LIN {X 0,Y 523.905,Z 250.039,A -85,B 0,C 180,E1 -4666.027,E2 -4666.027} C_VEL
LIN {X 0,Y 523.954,Z 250.034,A -85,B 0,C 180,E1 -4668.393,E2 -4668.393} C_VEL
LIN {X 0,Y 523.94,Z 250.032,A -85,B 0,C 180,E1 -4671.515,E2 -4671.515} C_VEL
LIN {X 0,Y 524.027,Z 250.021,A -85,B 0,C 180,E1 -4674.613,E2 -4674.613} C_VEL
LIN {X 0,Y 524.098,Z 250.015,A -85,B 0,C 180,E1 -4677.694,E2 -4677.694} C_VEL
LIN {X 0,Y 524.09,Z 250.017,A -85,B 0,C 180,E1 -4680,E2 -4680} C_VEL
LIN {X 0,Y 524.098,Z 250.013,A -85,B 0,C 180,E1 -4682.305,E2 -4682.305} C_VEL
LIN {X 0,Y 523.995,Z 250.027,A -85,B 0,C 180,E1 -4686.16,E2 -4686.16} C_VEL
LIN {X 0,Y 523.937,Z 250.033,A -85,B 0,C 180,E1 -4689.263,E2 -4689.263} C_VEL
LIN {X 0,Y 523.937,Z 250.031,A -85,B 0,C 180,E1 -4692.393,E2 -4692.393} C_VEL
LIN {X 0,Y 523.905,Z 250.04,A -85,B 0,C 180,E1 -4695.563,E2 -4695.563} C_VEL
LIN {X 0,Y 523.903,Z 250.037,A -85,B 0,C 180,E1 -4697.971,E2 -4697.971} C_VEL
LIN {X 0,Y 523.909,Z 250.033,A -85,B 0,C 180,E1 -4700.412,E2 -4700.412} C_VEL
LIN {X 0,Y 523.878,Z 250.039,A -85,B 0,C 180,E1 -4702.895,E2 -4702.895} C_VEL
LIN {X 0,Y 523.889,Z 250.043,A -85,B 0,C 180,E1 -4705.422,E2 -4705.422} C_VEL
LIN {X 0,Y 523.889,Z 250.037,A -85,B 0,C 180,E1 -4708.003,E2 -4708.003} C_VEL
LIN {X 0,Y 523.891,Z 250.039,A -85,B 0,C 180,E1 -4710.846,E2 -4710.846} C_VEL
LIN {X 0,Y 523.92,Z 250.034,A -85,B 0,C 180,E1 -4713.729,E2 -4713.729} C_VEL
LIN {X 0,Y 523.861,Z 250.04,A -85,B 0,C 180,E1 -4716.396,E2 -4716.396} C_VEL
LIN {X 0,Y 523.897,Z 250.042,A -85,B 0,C 180,E1 -4719.087,E2 -4719.087} C_VEL
LIN {X 0,Y 523.887,Z 250.036,A -85,B 0,C 180,E1 -4722.125,E2 -4722.125} C_VEL
LIN {X 0,Y 523.928,Z 250.035,A -85,B 0,C 180,E1 -4725.312,E2 -4725.312} C_VEL
LIN {X 0,Y 523.906,Z 250.038,A -85,B 0,C 180,E1 -4728.696,E2 -4728.696} C_VEL
LIN {X 0,Y 523.894,Z 250.035,A -85,B 0,C 180,E1 -4731.897,E2 -4731.897} C_VEL
LIN {X 0,Y 523.906,Z 250.04,A -85,B 0,C 180,E1 -4734.914,E2 -4734.914} C_VEL
LIN {X 0,Y 523.894,Z 250.034,A -85,B 0,C 180,E1 -4737.687,E2 -4737.687} C_VEL
LIN {X 0,Y 523.861,Z 250.041,A -85,B 0,C 180,E1 -4740.24,E2 -4740.24} C_VEL
LIN {X 0,Y 523.887,Z 250.042,A -85,B 0,C 180,E1 -4742.864,E2 -4742.864} C_VEL
LIN {X 0,Y 523.92,Z 250.04,A -85,B 0,C 180,E1 -4746.271,E2 -4746.271} C_VEL
LIN {X 0,Y 524.919,Z 256.867,A -85,B 0,C 180,E1 -4747.491,E2 -4747.491} C_VEL
LIN {X 0,Y 524.608,Z 272.008,A -85,B 0,C 180,E1 -4750.04,E2 -4750.04} C_VEL
LIN {X 0,Y 524.347,Z 287.74,A -85,B 0,C 180,E1 -4752.658,E2 -4752.658} C_VEL
LIN {X 0,Y 524.067,Z 307.036,A -85,B 0,C 180,E1 -4755.834,E2 -4755.834} C_VEL
LIN {X 0,Y 523.837,Z 320.787,A -85,B 0,C 180,E1 -4758.077,E2 -4758.077} C_VEL
LIN {X 0,Y 524.912,Z 332.835,A -85,B 0,C 180,E1 -4758.269,E2 -4758.269} C_VEL
LIN {X 0,Y 524.717,Z 397.742,A -85,B 0,C 180,E1 -4759.168,E2 -4759.168} C_VEL
LIN {X 0,Y 524.544,Z 407.017,A -85,B 0,C 180,E1 -4759.384,E2 -4759.384} C_VEL
LIN {X 0,Y 524.443,Z 415.51,A -85,B 0,C 180,E1 -4759.675,E2 -4759.675} C_VEL
LIN {X 0,Y 524.283,Z 424.041,A -85,B 0,C 180,E1 -4760.062,E2 -4760.062} C_VEL
LIN {X 0,Y 524.146,Z 432.41,A -85,B 0,C 180,E1 -4760.547,E2 -4760.547} C_VEL
LIN {X 0,Y 524.027,Z 440.49,A -85,B 0,C 180,E1 -4761.128,E2 -4761.128} C_VEL
LIN {X 0,Y 523.808,Z 449.21,A -85,B 0,C 180,E1 -4761.902,E2 -4761.902} C_VEL
LIN {X 0,Y 523.696,Z 457.778,A -85,B 0,C 180,E1 -4762.87,E2 -4762.87} C_VEL
LIN {X 0,Y 523.586,Z 464.502,A -85,B 0,C 180,E1 -4763.836,E2 -4763.836} C_VEL
LIN {X 0,Y 523.483,Z 468.916,A -85,B 0,C 180,E1 -4764.608,E2 -4764.608} C_VEL
LIN {X 0,Y 523.45,Z 474.125,A -85,B 0,C 180,E1 -4765.766,E2 -4765.766} C_VEL
LIN {X 0,Y 523.406,Z 476.787,A -85,B 0,C 180,E1 -4766.536,E2 -4766.536} C_VEL
LIN {X 0,Y 523.336,Z 479.706,A -85,B 0,C 180,E1 -4767.691,E2 -4767.691} C_VEL
LIN {X 0,Y 523.273,Z 480.964,A -85,B 0,C 180,E1 -4768.461,E2 -4768.461} C_VEL
LIN {X 0,Y 523.26,Z 481.749,A -85,B 0,C 180,E1 -4769.231,E2 -4769.231} C_VEL
LIN {X 0,Y 523.264,Z 482.046,A -85,B 0,C 180,E1 -4770,E2 -4770} C_VEL
LIN {X 0,Y 523.26,Z 481.748,A -85,B 0,C 180,E1 -4770.77,E2 -4770.77} C_VEL
LIN {X 0,Y 523.273,Z 480.963,A -85,B 0,C 180,E1 -4771.54,E2 -4771.54} C_VEL
LIN {X 0,Y 523.336,Z 479.704,A -85,B 0,C 180,E1 -4772.309,E2 -4772.309} C_VEL
LIN {X 0,Y 523.407,Z 476.784,A -85,B 0,C 180,E1 -4773.464,E2 -4773.464} C_VEL
LIN {X 0,Y 523.451,Z 474.122,A -85,B 0,C 180,E1 -4774.235,E2 -4774.235} C_VEL
LIN {X 0,Y 523.483,Z 468.909,A -85,B 0,C 180,E1 -4775.393,E2 -4775.393} C_VEL
LIN {X 0,Y 523.573,Z 462.995,A -85,B 0,C 180,E1 -4776.409,E2 -4776.409} C_VEL
LIN {X 0,Y 523.699,Z 456.256,A -85,B 0,C 180,E1 -4777.325,E2 -4777.325} C_VEL
LIN {X 0,Y 523.833,Z 448.182,A -85,B 0,C 180,E1 -4778.196,E2 -4778.196} C_VEL
LIN {X 0,Y 524.028,Z 440.484,A -85,B 0,C 180,E1 -4778.873,E2 -4778.873} C_VEL
LIN {X 0,Y 524.147,Z 432.399,A -85,B 0,C 180,E1 -4779.454,E2 -4779.454} C_VEL
LIN {X 0,Y 524.283,Z 424.028,A -85,B 0,C 180,E1 -4779.939,E2 -4779.939} C_VEL
LIN {X 0,Y 524.443,Z 415.494,A -85,B 0,C 180,E1 -4780.326,E2 -4780.326} C_VEL
LIN {X 0,Y 524.588,Z 405.328,A -85,B 0,C 180,E1 -4780.664,E2 -4780.664} C_VEL
LIN {X 0,Y 524.728,Z 393.603,A -85,B 0,C 180,E1 -4780.906,E2 -4780.906} C_VEL
LIN {X 0,Y 524.84,Z 329.868,A -85,B 0,C 180,E1 -4781.773,E2 -4781.773} C_VEL
LIN {X 0,Y 523.822,Z 320.739,A -85,B 0,C 180,E1 -4781.931,E2 -4781.931} C_VEL
LIN {X 0,Y 524.065,Z 303.407,A -85,B 0,C 180,E1 -4784.762,E2 -4784.762} C_VEL
LIN {X 0,Y 524.416,Z 284.047,A -85,B 0,C 180,E1 -4787.953,E2 -4787.953} C_VEL
LIN {X 0,Y 524.723,Z 265.839,A -85,B 0,C 180,E1 -4790.995,E2 -4790.995} C_VEL
LIN {X 0,Y 524.885,Z 256.204,A -85,B 0,C 180,E1 -4792.623,E2 -4792.623} C_VEL
LIN {X 0,Y 523.923,Z 250.038,A -85,B 0,C 180,E1 -4793.73,E2 -4793.73} C_VEL
LIN {X 0,Y 523.89,Z 250.042,A -85,B 0,C 180,E1 -4797.137,E2 -4797.137} C_VEL
LIN {X 0,Y 523.865,Z 250.041,A -85,B 0,C 180,E1 -4799.761,E2 -4799.761} C_VEL
LIN {X 0,Y 523.895,Z 250.034,A -85,B 0,C 180,E1 -4802.453,E2 -4802.453} C_VEL
LIN {X 0,Y 523.88,Z 250.045,A -85,B 0,C 180,E1 -4805.23,E2 -4805.23} C_VEL
LIN {X 0,Y 523.877,Z 250.037,A -85,B 0,C 180,E1 -4808.105,E2 -4808.105} C_VEL
LIN {X 0,Y 523.88,Z 250.042,A -85,B 0,C 180,E1 -4811.301,E2 -4811.301} C_VEL
LIN {X 0,Y 523.932,Z 250.034,A -85,B 0,C 180,E1 -4814.689,E2 -4814.689} C_VEL
LIN {X 0,Y 523.889,Z 250.035,A -85,B 0,C 180,E1 -4817.875,E2 -4817.875} C_VEL
LIN {X 0,Y 523.894,Z 250.042,A -85,B 0,C 180,E1 -4820.913,E2 -4820.913} C_VEL
LIN {X 0,Y 523.853,Z 250.04,A -85,B 0,C 180,E1 -4823.822,E2 -4823.822} C_VEL
LIN {X 0,Y 523.895,Z 250.041,A -85,B 0,C 180,E1 -4826.632,E2 -4826.632} C_VEL
LIN {X 0,Y 523.906,Z 250.035,A -85,B 0,C 180,E1 -4829.353,E2 -4829.353} C_VEL
LIN {X 0,Y 523.911,Z 250.037,A -85,B 0,C 180,E1 -4832.296,E2 -4832.296} C_VEL
LIN {X 0,Y 523.89,Z 250.036,A -85,B 0,C 180,E1 -4835.426,E2 -4835.426} C_VEL
LIN {X 0,Y 523.92,Z 250.033,A -85,B 0,C 180,E1 -4837.939,E2 -4837.939} C_VEL
LIN {X 0,Y 523.9,Z 250.042,A -85,B 0,C 180,E1 -4840.405,E2 -4840.405} C_VEL
LIN {X 0,Y 523.9,Z 250.038,A -85,B 0,C 180,E1 -4842.835,E2 -4842.835} C_VEL
LIN {X 0,Y 523.92,Z 250.032,A -85,B 0,C 180,E1 -4845.234,E2 -4845.234} C_VEL
LIN {X 0,Y 523.96,Z 250.033,A -85,B 0,C 180,E1 -4848.393,E2 -4848.393} C_VEL
LIN {X 0,Y 523.945,Z 250.03,A -85,B 0,C 180,E1 -4851.515,E2 -4851.515} C_VEL
LIN {X 0,Y 524.028,Z 250.023,A -85,B 0,C 180,E1 -4854.613,E2 -4854.613} C_VEL
LIN {X 0,Y 524.103,Z 250.012,A -85,B 0,C 180,E1 -4857.695,E2 -4857.695} C_VEL
LIN {X 0,Y 524.096,Z 250.017,A -85,B 0,C 180,E1 -4860,E2 -4860} C_VEL
LIN {X 0,Y 524.103,Z 250.014,A -85,B 0,C 180,E1 -4862.306,E2 -4862.306} C_VEL
LIN {X 0,Y 524.001,Z 250.027,A -85,B 0,C 180,E1 -4866.16,E2 -4866.16} C_VEL
LIN {X 0,Y 523.944,Z 250.031,A -85,B 0,C 180,E1 -4869.263,E2 -4869.263} C_VEL
LIN {X 0,Y 523.945,Z 250.032,A -85,B 0,C 180,E1 -4872.393,E2 -4872.393} C_VEL
LIN {X 0,Y 523.913,Z 250.039,A -85,B 0,C 180,E1 -4875.563,E2 -4875.563} C_VEL
LIN {X 0,Y 523.911,Z 250.039,A -85,B 0,C 180,E1 -4877.971,E2 -4877.971} C_VEL
LIN {X 0,Y 523.917,Z 250.034,A -85,B 0,C 180,E1 -4880.412,E2 -4880.412} C_VEL
LIN {X 0,Y 523.885,Z 250.038,A -85,B 0,C 180,E1 -4882.895,E2 -4882.895} C_VEL
LIN {X 0,Y 523.899,Z 250.041,A -85,B 0,C 180,E1 -4885.422,E2 -4885.422} C_VEL
LIN {X 0,Y 523.897,Z 250.038,A -85,B 0,C 180,E1 -4888.003,E2 -4888.003} C_VEL
LIN {X 0,Y 523.902,Z 250.036,A -85,B 0,C 180,E1 -4890.846,E2 -4890.846} C_VEL
LIN {X 0,Y 523.927,Z 250.036,A -85,B 0,C 180,E1 -4893.729,E2 -4893.729} C_VEL
LIN {X 0,Y 523.888,Z 250.037,A -85,B 0,C 180,E1 -4896.399,E2 -4896.399} C_VEL
LIN {X 0,Y 523.91,Z 250.039,A -85,B 0,C 180,E1 -4899.086,E2 -4899.086} C_VEL
LIN {X 0,Y 523.893,Z 250.036,A -85,B 0,C 180,E1 -4902.125,E2 -4902.125} C_VEL
LIN {X 0,Y 523.935,Z 250.036,A -85,B 0,C 180,E1 -4905.311,E2 -4905.311} C_VEL
LIN {X 0,Y 523.879,Z 250.042,A -85,B 0,C 180,E1 -4906.868,E2 -4906.868} C_VEL
LIN {X 0,Y 523.192,Z 250.127,A -85,B 0,C 180,E1 -4907.51,E2 -4907.51} C_VEL
LIN {X 0,Y 520.329,Z 250.482,A -85,B 0,C 180,E1 -4908.551,E2 -4908.551} C_VEL
LIN {X 0,Y 517.935,Z 250.783,A -85,B 0,C 180,E1 -4909.39,E2 -4909.39} C_VEL
LIN {X 0,Y 516.929,Z 250.904,A -85,B 0,C 180,E1 -4910.038,E2 -4910.038} C_VEL
LIN {X 0,Y 516.858,Z 250.913,A -85,B 0,C 180,E1 -4910.257,E2 -4910.257} C_VEL
LIN {X 0,Y 516.854,Z 250.919,A -85,B 0,C 180,E1 -4913.252,E2 -4913.252} C_VEL
LIN {X 0,Y 516.881,Z 250.91,A -85,B 0,C 180,E1 -4916.118,E2 -4916.118} C_VEL
LIN {X 0,Y 516.85,Z 250.919,A -85,B 0,C 180,E1 -4918.944,E2 -4918.944} C_VEL
LIN {X 0,Y 516.846,Z 250.915,A -85,B 0,C 180,E1 -4921.58,E2 -4921.58} C_VEL
LIN {X 0,Y 516.871,Z 250.912,A -85,B 0,C 180,E1 -4924.207,E2 -4924.207} C_VEL
LIN {X 0,Y 516.853,Z 250.918,A -85,B 0,C 180,E1 -4926.775,E2 -4926.775} C_VEL
LIN {X 0,Y 516.929,Z 250.903,A -85,B 0,C 180,E1 -4929.735,E2 -4929.735} C_VEL
LIN {X 0,Y 516.879,Z 250.917,A -85,B 0,C 180,E1 -4932.594,E2 -4932.594} C_VEL
LIN {X 0,Y 516.693,Z 250.994,A -85,B 0,C 180,E1 -4934.548,E2 -4934.548} C_VEL
LIN {X 0,Y 516.644,Z 265.328,A -85,B 0,C 180,E1 -4937.788,E2 -4937.788} C_VEL
LIN {X 0,Y 516.655,Z 266.191,A -85,B 0,C 180,E1 -4937.977,E2 -4937.977} C_VEL
LIN {X 0,Y 518.082,Z 276.255,A -85,B 0,C 180,E1 -4938.154,E2 -4938.154} C_VEL
LIN {X 0,Y 517.773,Z 341.417,A -85,B 0,C 180,E1 -4939.07,E2 -4939.07} C_VEL
LIN {X 0,Y 517.698,Z 349.767,A -85,B 0,C 180,E1 -4939.266,E2 -4939.266} C_VEL
LIN {X 0,Y 517.58,Z 359.014,A -85,B 0,C 180,E1 -4939.585,E2 -4939.585} C_VEL
LIN {X 0,Y 517.478,Z 366.536,A -85,B 0,C 180,E1 -4939.929,E2 -4939.929} C_VEL
LIN {X 0,Y 517.334,Z 375.007,A -85,B 0,C 180,E1 -4940.42,E2 -4940.42} C_VEL
LIN {X 0,Y 517.215,Z 383.133,A -85,B 0,C 180,E1 -4941.01,E2 -4941.01} C_VEL
LIN {X 0,Y 517.03,Z 390.845,A -85,B 0,C 180,E1 -4941.696,E2 -4941.696} C_VEL
LIN {X 0,Y 516.857,Z 397.209,A -85,B 0,C 180,E1 -4942.381,E2 -4942.381} C_VEL
LIN {X 0,Y 516.724,Z 404.187,A -85,B 0,C 180,E1 -4943.293,E2 -4943.293} C_VEL
LIN {X 0,Y 516.5,Z 410.57,A -85,B 0,C 180,E1 -4944.338,E2 -4944.338} C_VEL
LIN {X 0,Y 516.512,Z 415.188,A -85,B 0,C 180,E1 -4945.317,E2 -4945.317} C_VEL
LIN {X 0,Y 516.391,Z 418.177,A -85,B 0,C 180,E1 -4946.098,E2 -4946.098} C_VEL
LIN {X 0,Y 516.403,Z 420.488,A -85,B 0,C 180,E1 -4946.879,E2 -4946.879} C_VEL
LIN {X 0,Y 516.269,Z 422.26,A -85,B 0,C 180,E1 -4947.659,E2 -4947.659} C_VEL
LIN {X 0,Y 516.2,Z 423.537,A -85,B 0,C 180,E1 -4948.439,E2 -4948.439} C_VEL
LIN {X 0,Y 516.186,Z 424.345,A -85,B 0,C 180,E1 -4949.219,E2 -4949.219} C_VEL
LIN {X 0,Y 516.186,Z 424.653,A -85,B 0,C 180,E1 -4950,E2 -4950} C_VEL
LIN {X 0,Y 516.186,Z 424.383,A -85,B 0,C 180,E1 -4950.78,E2 -4950.78} C_VEL
LIN {X 0,Y 516.201,Z 423.649,A -85,B 0,C 180,E1 -4951.56,E2 -4951.56} C_VEL
LIN {X 0,Y 516.269,Z 422.447,A -85,B 0,C 180,E1 -4952.34,E2 -4952.34} C_VEL
LIN {X 0,Y 516.418,Z 419.614,A -85,B 0,C 180,E1 -4953.511,E2 -4953.511} C_VEL
LIN {X 0,Y 516.433,Z 417.043,A -85,B 0,C 180,E1 -4954.292,E2 -4954.292} C_VEL
LIN {X 0,Y 516.433,Z 411.976,A -85,B 0,C 180,E1 -4955.466,E2 -4955.466} C_VEL
LIN {X 0,Y 516.703,Z 405.867,A -85,B 0,C 180,E1 -4956.55,E2 -4956.55} C_VEL
LIN {X 0,Y 516.854,Z 397.988,A -85,B 0,C 180,E1 -4957.618,E2 -4957.618} C_VEL
LIN {X 0,Y 516.995,Z 390.762,A -85,B 0,C 180,E1 -4958.403,E2 -4958.403} C_VEL
LIN {X 0,Y 517.203,Z 384.256,A -85,B 0,C 180,E1 -4958.99,E2 -4958.99} C_VEL
LIN {X 0,Y 517.3,Z 376.382,A -85,B 0,C 180,E1 -4959.58,E2 -4959.58} C_VEL
LIN {X 0,Y 517.484,Z 368.247,A -85,B 0,C 180,E1 -4960.07,E2 -4960.07} C_VEL
LIN {X 0,Y 517.611,Z 360.017,A -85,B 0,C 180,E1 -4960.463,E2 -4960.463} C_VEL
LIN {X 0,Y 517.677,Z 351.151,A -85,B 0,C 180,E1 -4960.783,E2 -4960.783} C_VEL
LIN {X 0,Y 517.866,Z 342.414,A -85,B 0,C 180,E1 -4960.999,E2 -4960.999} C_VEL
LIN {X 0,Y 518.009,Z 295.646,A -85,B 0,C 180,E1 -4961.669,E2 -4961.669} C_VEL
LIN {X 0,Y 518.006,Z 274.632,A -85,B 0,C 180,E1 -4961.961,E2 -4961.961} C_VEL
LIN {X 0,Y 516.658,Z 266.136,A -85,B 0,C 180,E1 -4962.127,E2 -4962.127} C_VEL
LIN {X 0,Y 516.663,Z 251.854,A -85,B 0,C 180,E1 -4965.341,E2 -4965.341} C_VEL
LIN {X 0,Y 516.672,Z 250.945,A -85,B 0,C 180,E1 -4965.563,E2 -4965.563} C_VEL
LIN {X 0,Y 516.873,Z 250.914,A -85,B 0,C 180,E1 -4967.861,E2 -4967.861} C_VEL
LIN {X 0,Y 516.889,Z 250.909,A -85,B 0,C 180,E1 -4970.702,E2 -4970.702} C_VEL
LIN {X 0,Y 516.838,Z 250.921,A -85,B 0,C 180,E1 -4973.224,E2 -4973.224} C_VEL
LIN {X 0,Y 516.879,Z 250.91,A -85,B 0,C 180,E1 -4976.181,E2 -4976.181} C_VEL
LIN {X 0,Y 516.895,Z 250.913,A -85,B 0,C 180,E1 -4979.306,E2 -4979.306} C_VEL
LIN {X 0,Y 516.889,Z 250.91,A -85,B 0,C 180,E1 -4982.542,E2 -4982.542} C_VEL
LIN {X 0,Y 516.851,Z 250.918,A -85,B 0,C 180,E1 -4985.327,E2 -4985.327} C_VEL
LIN {X 0,Y 516.874,Z 250.911,A -85,B 0,C 180,E1 -4987.942,E2 -4987.942} C_VEL
LIN {X 0,Y 516.846,Z 250.92,A -85,B 0,C 180,E1 -4990.744,E2 -4990.744} C_VEL
LIN {X 0,Y 516.876,Z 250.91,A -85,B 0,C 180,E1 -4993.903,E2 -4993.903} C_VEL
LIN {X 0,Y 516.876,Z 250.911,A -85,B 0,C 180,E1 -4996.107,E2 -4996.107} C_VEL
LIN {X 0,Y 516.843,Z 250.917,A -85,B 0,C 180,E1 -4999.254,E2 -4999.254} C_VEL
LIN {X 0,Y 516.871,Z 250.912,A -85,B 0,C 180,E1 -5002.057,E2 -5002.057} C_VEL
LIN {X 0,Y 516.866,Z 250.914,A -85,B 0,C 180,E1 -5005.174,E2 -5005.174} C_VEL
LIN {X 0,Y 516.861,Z 250.913,A -85,B 0,C 180,E1 -5007.974,E2 -5007.974} C_VEL
LIN {X 0,Y 516.892,Z 250.913,A -85,B 0,C 180,E1 -5010.694,E2 -5010.694} C_VEL
LIN {X 0,Y 516.874,Z 250.912,A -85,B 0,C 180,E1 -5013.818,E2 -5013.818} C_VEL
LIN {X 0,Y 516.836,Z 250.919,A -85,B 0,C 180,E1 -5016.775,E2 -5016.775} C_VEL
LIN {X 0,Y 516.901,Z 250.909,A -85,B 0,C 180,E1 -5019.742,E2 -5019.742} C_VEL
LIN {X 0,Y 516.873,Z 250.915,A -85,B 0,C 180,E1 -5022.594,E2 -5022.594} C_VEL
LIN {X 0,Y 516.925,Z 250.905,A -85,B 0,C 180,E1 -5025.03,E2 -5025.03} C_VEL
LIN {X 0,Y 516.92,Z 250.91,A -85,B 0,C 180,E1 -5028.233,E2 -5028.233} C_VEL
LIN {X 0,Y 516.914,Z 250.906,A -85,B 0,C 180,E1 -5031.399,E2 -5031.399} C_VEL
LIN {X 0,Y 516.978,Z 250.9,A -85,B 0,C 180,E1 -5034.539,E2 -5034.539} C_VEL
LIN {X 0,Y 517.067,Z 250.891,A -85,B 0,C 180,E1 -5037.663,E2 -5037.663} C_VEL
LIN {X 0,Y 517.059,Z 250.893,A -85,B 0,C 180,E1 -5040,E2 -5040} C_VEL
LIN {X 0,Y 517.067,Z 250.889,A -85,B 0,C 180,E1 -5042.337,E2 -5042.337} C_VEL
LIN {X 0,Y 516.962,Z 250.902,A -85,B 0,C 180,E1 -5046.244,E2 -5046.244} C_VEL
LIN {X 0,Y 516.9,Z 250.911,A -85,B 0,C 180,E1 -5049.39,E2 -5049.39} C_VEL
LIN {X 0,Y 516.89,Z 250.908,A -85,B 0,C 180,E1 -5052.565,E2 -5052.565} C_VEL
LIN {X 0,Y 516.929,Z 250.906,A -85,B 0,C 180,E1 -5055.142,E2 -5055.142} C_VEL
LIN {X 0,Y 516.863,Z 250.912,A -85,B 0,C 180,E1 -5058.224,E2 -5058.224} C_VEL
LIN {X 0,Y 516.864,Z 250.912,A -85,B 0,C 180,E1 -5060.703,E2 -5060.703} C_VEL
LIN {X 0,Y 516.833,Z 250.919,A -85,B 0,C 180,E1 -5063.225,E2 -5063.225} C_VEL
LIN {X 0,Y 516.872,Z 250.91,A -85,B 0,C 180,E1 -5066.181,E2 -5066.181} C_VEL
LIN {X 0,Y 516.822,Z 250.916,A -85,B 0,C 180,E1 -5068.421,E2 -5068.421} C_VEL
LIN {X 0,Y 516.842,Z 250.919,A -85,B 0,C 180,E1 -5071.113,E2 -5071.113} C_VEL
LIN {X 0,Y 516.874,Z 250.91,A -85,B 0,C 180,E1 -5073.962,E2 -5073.962} C_VEL
LIN {X 0,Y 516.809,Z 250.921,A -85,B 0,C 180,E1 -5076.752,E2 -5076.752} C_VEL
LIN {X 0,Y 516.85,Z 250.914,A -85,B 0,C 180,E1 -5079.724,E2 -5079.724} C_VEL
LIN {X 0,Y 516.836,Z 250.919,A -85,B 0,C 180,E1 -5082.836,E2 -5082.836} C_VEL
LIN {X 0,Y 516.891,Z 250.915,A -85,B 0,C 180,E1 -5085.007,E2 -5085.007} C_VEL
LIN {X 0,Y 516.844,Z 250.915,A -85,B 0,C 180,E1 -5088.407,E2 -5088.407} C_VEL
LIN {X 0,Y 516.864,Z 250.913,A -85,B 0,C 180,E1 -5091.283,E2 -5091.283} C_VEL
LIN {X 0,Y 516.843,Z 250.919,A -85,B 0,C 180,E1 -5094.674,E2 -5094.674} C_VEL
LIN {X 0,Y 516.859,Z 250.911,A -85,B 0,C 180,E1 -5097.463,E2 -5097.463} C_VEL
LIN {X 0,Y 516.834,Z 250.92,A -85,B 0,C 180,E1 -5100.491,E2 -5100.491} C_VEL
LIN {X 0,Y 516.824,Z 250.917,A -85,B 0,C 180,E1 -5103.337,E2 -5103.337} C_VEL
LIN {X 0,Y 516.892,Z 251.08,A -85,B 0,C 180,E1 -5106.194,E2 -5106.194} C_VEL
LIN {X 0,Y 517.895,Z 257.448,A -85,B 0,C 180,E1 -5107.336,E2 -5107.336} C_VEL
LIN {X 0,Y 517.628,Z 272.083,A -85,B 0,C 180,E1 -5109.836,E2 -5109.836} C_VEL
LIN {X 0,Y 517.32,Z 288.522,A -85,B 0,C 180,E1 -5112.61,E2 -5112.61} C_VEL
LIN {X 0,Y 517.012,Z 307.855,A -85,B 0,C 180,E1 -5115.837,E2 -5115.837} C_VEL
LIN {X 0,Y 516.782,Z 320.362,A -85,B 0,C 180,E1 -5117.908,E2 -5117.908} C_VEL
LIN {X 0,Y 517.96,Z 333.268,A -85,B 0,C 180,E1 -5118.12,E2 -5118.12} C_VEL
LIN {X 0,Y 517.722,Z 397.372,A -85,B 0,C 180,E1 -5119.021,E2 -5119.021} C_VEL
LIN {X 0,Y 517.563,Z 406.625,A -85,B 0,C 180,E1 -5119.24,E2 -5119.24} C_VEL
LIN {X 0,Y 517.454,Z 415.118,A -85,B 0,C 180,E1 -5119.534,E2 -5119.534} C_VEL
LIN {X 0,Y 517.269,Z 423.648,A -85,B 0,C 180,E1 -5119.926,E2 -5119.926} C_VEL
LIN {X 0,Y 517.12,Z 432.017,A -85,B 0,C 180,E1 -5120.417,E2 -5120.417} C_VEL
LIN {X 0,Y 516.946,Z 440.094,A -85,B 0,C 180,E1 -5121.006,E2 -5121.006} C_VEL
LIN {X 0,Y 516.751,Z 447.789,A -85,B 0,C 180,E1 -5121.692,E2 -5121.692} C_VEL
LIN {X 0,Y 516.622,Z 455.868,A -85,B 0,C 180,E1 -5122.575,E2 -5122.575} C_VEL
LIN {X 0,Y 516.483,Z 463.243,A -85,B 0,C 180,E1 -5123.608,E2 -5123.608} C_VEL
LIN {X 0,Y 516.42,Z 468.525,A -85,B 0,C 180,E1 -5124.534,E2 -5124.534} C_VEL
LIN {X 0,Y 516.358,Z 473.733,A -85,B 0,C 180,E1 -5125.707,E2 -5125.707} C_VEL
LIN {X 0,Y 516.324,Z 476.395,A -85,B 0,C 180,E1 -5126.489,E2 -5126.489} C_VEL
LIN {X 0,Y 516.262,Z 479.315,A -85,B 0,C 180,E1 -5127.66,E2 -5127.66} C_VEL
LIN {X 0,Y 516.19,Z 480.573,A -85,B 0,C 180,E1 -5128.44,E2 -5128.44} C_VEL
LIN {X 0,Y 516.171,Z 481.357,A -85,B 0,C 180,E1 -5129.22,E2 -5129.22} C_VEL
LIN {X 0,Y 516.175,Z 481.655,A -85,B 0,C 180,E1 -5130,E2 -5130} C_VEL
LIN {X 0,Y 516.171,Z 481.357,A -85,B 0,C 180,E1 -5130.781,E2 -5130.781} C_VEL
LIN {X 0,Y 516.19,Z 480.571,A -85,B 0,C 180,E1 -5131.561,E2 -5131.561} C_VEL
LIN {X 0,Y 516.263,Z 479.313,A -85,B 0,C 180,E1 -5132.341,E2 -5132.341} C_VEL
LIN {X 0,Y 516.324,Z 476.392,A -85,B 0,C 180,E1 -5133.512,E2 -5133.512} C_VEL
LIN {X 0,Y 516.358,Z 473.729,A -85,B 0,C 180,E1 -5134.293,E2 -5134.293} C_VEL
LIN {X 0,Y 516.42,Z 468.518,A -85,B 0,C 180,E1 -5135.467,E2 -5135.467} C_VEL
LIN {X 0,Y 516.476,Z 463.28,A -85,B 0,C 180,E1 -5136.385,E2 -5136.385} C_VEL
LIN {X 0,Y 516.623,Z 455.862,A -85,B 0,C 180,E1 -5137.426,E2 -5137.426} C_VEL
LIN {X 0,Y 516.752,Z 447.787,A -85,B 0,C 180,E1 -5138.309,E2 -5138.309} C_VEL
LIN {X 0,Y 516.947,Z 440.088,A -85,B 0,C 180,E1 -5138.995,E2 -5138.995} C_VEL
LIN {X 0,Y 517.12,Z 432.005,A -85,B 0,C 180,E1 -5139.584,E2 -5139.584} C_VEL
LIN {X 0,Y 517.269,Z 423.635,A -85,B 0,C 180,E1 -5140.075,E2 -5140.075} C_VEL
LIN {X 0,Y 517.455,Z 415.101,A -85,B 0,C 180,E1 -5140.467,E2 -5140.467} C_VEL
LIN {X 0,Y 517.586,Z 405.768,A -85,B 0,C 180,E1 -5140.786,E2 -5140.786} C_VEL
LIN {X 0,Y 517.745,Z 394.812,A -85,B 0,C 180,E1 -5141.028,E2 -5141.028} C_VEL
LIN {X 0,Y 517.866,Z 330.307,A -85,B 0,C 180,E1 -5141.923,E2 -5141.923} C_VEL
LIN {X 0,Y 516.795,Z 320.319,A -85,B 0,C 180,E1 -5142.099,E2 -5142.099} C_VEL
LIN {X 0,Y 517.011,Z 303.02,A -85,B 0,C 180,E1 -5144.968,E2 -5144.968} C_VEL
LIN {X 0,Y 517.481,Z 282.464,A -85,B 0,C 180,E1 -5148.407,E2 -5148.407} C_VEL
LIN {X 0,Y 517.747,Z 264.242,A -85,B 0,C 180,E1 -5151.5,E2 -5151.5} C_VEL
LIN {X 0,Y 517.801,Z 256.264,A -85,B 0,C 180,E1 -5152.872,E2 -5152.872} C_VEL
LIN {X 0,Y 516.868,Z 250.915,A -85,B 0,C 180,E1 -5153.861,E2 -5153.861} C_VEL
LIN {X 0,Y 516.827,Z 250.917,A -85,B 0,C 180,E1 -5156.664,E2 -5156.664} C_VEL
LIN {X 0,Y 516.837,Z 250.92,A -85,B 0,C 180,E1 -5159.509,E2 -5159.509} C_VEL
LIN {X 0,Y 516.863,Z 250.911,A -85,B 0,C 180,E1 -5162.538,E2 -5162.538} C_VEL
LIN {X 0,Y 516.826,Z 250.922,A -85,B 0,C 180,E1 -5165.323,E2 -5165.323} C_VEL
LIN {X 0,Y 516.854,Z 250.914,A -85,B 0,C 180,E1 -5168.719,E2 -5168.719} C_VEL
LIN {X 0,Y 516.832,Z 250.915,A -85,B 0,C 180,E1 -5171.783,E2 -5171.783} C_VEL
LIN {X 0,Y 516.896,Z 250.914,A -85,B 0,C 180,E1 -5175.007,E2 -5175.007} C_VEL
LIN {X 0,Y 516.847,Z 250.915,A -85,B 0,C 180,E1 -5178.407,E2 -5178.407} C_VEL
LIN {X 0,Y 516.859,Z 250.915,A -85,B 0,C 180,E1 -5181.282,E2 -5181.282} C_VEL
LIN {X 0,Y 516.847,Z 250.919,A -85,B 0,C 180,E1 -5184.674,E2 -5184.674} C_VEL
LIN {X 0,Y 516.863,Z 250.912,A -85,B 0,C 180,E1 -5187.463,E2 -5187.463} C_VEL
LIN {X 0,Y 516.837,Z 250.92,A -85,B 0,C 180,E1 -5190.491,E2 -5190.491} C_VEL
LIN {X 0,Y 516.828,Z 250.917,A -85,B 0,C 180,E1 -5193.337,E2 -5193.337} C_VEL
LIN {X 0,Y 516.857,Z 250.913,A -85,B 0,C 180,E1 -5195.925,E2 -5195.925} C_VEL
LIN {X 0,Y 516.849,Z 250.92,A -85,B 0,C 180,E1 -5198.461,E2 -5198.461} C_VEL
LIN {X 0,Y 516.845,Z 250.916,A -85,B 0,C 180,E1 -5200.953,E2 -5200.953} C_VEL
LIN {X 0,Y 516.832,Z 250.915,A -85,B 0,C 180,E1 -5203.408,E2 -5203.408} C_VEL
LIN {X 0,Y 516.848,Z 250.915,A -85,B 0,C 180,E1 -5205.832,E2 -5205.832} C_VEL
LIN {X 0,Y 516.92,Z 250.911,A -85,B 0,C 180,E1 -5208.233,E2 -5208.233} C_VEL
LIN {X 0,Y 516.919,Z 250.905,A -85,B 0,C 180,E1 -5211.399,E2 -5211.399} C_VEL
LIN {X 0,Y 516.979,Z 250.901,A -85,B 0,C 180,E1 -5214.54,E2 -5214.54} C_VEL
LIN {X 0,Y 517.072,Z 250.888,A -85,B 0,C 180,E1 -5217.663,E2 -5217.663} C_VEL
LIN {X 0,Y 517.065,Z 250.893,A -85,B 0,C 180,E1 -5220,E2 -5220} C_VEL
LIN {X 0,Y 517.073,Z 250.89,A -85,B 0,C 180,E1 -5222.337,E2 -5222.337} C_VEL
LIN {X 0,Y 516.968,Z 250.903,A -85,B 0,C 180,E1 -5226.244,E2 -5226.244} C_VEL
LIN {X 0,Y 516.907,Z 250.908,A -85,B 0,C 180,E1 -5229.39,E2 -5229.39} C_VEL
LIN {X 0,Y 516.897,Z 250.908,A -85,B 0,C 180,E1 -5232.565,E2 -5232.565} C_VEL
LIN {X 0,Y 516.937,Z 250.904,A -85,B 0,C 180,E1 -5235.142,E2 -5235.142} C_VEL
LIN {X 0,Y 516.871,Z 250.913,A -85,B 0,C 180,E1 -5238.224,E2 -5238.224} C_VEL
LIN {X 0,Y 516.872,Z 250.911,A -85,B 0,C 180,E1 -5240.703,E2 -5240.703} C_VEL
LIN {X 0,Y 516.841,Z 250.918,A -85,B 0,C 180,E1 -5243.225,E2 -5243.225} C_VEL
LIN {X 0,Y 516.88,Z 250.911,A -85,B 0,C 180,E1 -5246.181,E2 -5246.181} C_VEL
LIN {X 0,Y 516.89,Z 250.914,A -85,B 0,C 180,E1 -5249.307,E2 -5249.307} C_VEL
LIN {X 0,Y 516.893,Z 250.908,A -85,B 0,C 180,E1 -5252.542,E2 -5252.542} C_VEL
LIN {X 0,Y 516.855,Z 250.918,A -85,B 0,C 180,E1 -5255.328,E2 -5255.328} C_VEL
LIN {X 0,Y 516.877,Z 250.912,A -85,B 0,C 180,E1 -5257.942,E2 -5257.942} C_VEL
LIN {X 0,Y 516.848,Z 250.916,A -85,B 0,C 180,E1 -5260.745,E2 -5260.745} C_VEL
LIN {X 0,Y 516.881,Z 250.911,A -85,B 0,C 180,E1 -5263.903,E2 -5263.903} C_VEL
LIN {X 0,Y 516.836,Z 250.917,A -85,B 0,C 180,E1 -5266.868,E2 -5266.868} C_VEL
LIN {X 0,Y 516.86,Z 250.915,A -85,B 0,C 180,E1 -5269.593,E2 -5269.593} C_VEL
LIN {X 0,Y 516.858,Z 250.913,A -85,B 0,C 180,E1 -5270.257,E2 -5270.257} C_VEL
LIN {X 0,Y 516.221,Z 250.996,A -85,B 0,C 180,E1 -5270.907,E2 -5270.907} C_VEL
LIN {X 0,Y 513.377,Z 251.352,A -85,B 0,C 180,E1 -5271.963,E2 -5271.963} C_VEL
LIN {X 0,Y 510.949,Z 251.654,A -85,B 0,C 180,E1 -5272.813,E2 -5272.813} C_VEL
LIN {X 0,Y 509.897,Z 251.783,A -85,B 0,C 180,E1 -5273.47,E2 -5273.47} C_VEL
LIN {X 0,Y 509.808,Z 251.792,A -85,B 0,C 180,E1 -5273.692,E2 -5273.692} C_VEL
LIN {X 0,Y 509.84,Z 251.79,A -85,B 0,C 180,E1 -5276.537,E2 -5276.537} C_VEL
LIN {X 0,Y 509.806,Z 251.794,A -85,B 0,C 180,E1 -5279.331,E2 -5279.331} C_VEL
LIN {X 0,Y 509.832,Z 251.788,A -85,B 0,C 180,E1 -5282.051,E2 -5282.051} C_VEL
LIN {X 0,Y 509.802,Z 251.796,A -85,B 0,C 180,E1 -5284.7,E2 -5284.7} C_VEL
LIN {X 0,Y 509.826,Z 251.789,A -85,B 0,C 180,E1 -5287.459,E2 -5287.459} C_VEL
LIN {X 0,Y 509.907,Z 251.779,A -85,B 0,C 180,E1 -5289.844,E2 -5289.844} C_VEL
LIN {X 0,Y 509.853,Z 251.79,A -85,B 0,C 180,E1 -5292.346,E2 -5292.346} C_VEL
LIN {X 0,Y 509.638,Z 251.865,A -85,B 0,C 180,E1 -5294.554,E2 -5294.554} C_VEL
LIN {X 0,Y 509.593,Z 265.539,A -85,B 0,C 180,E1 -5297.616,E2 -5297.616} C_VEL
LIN {X 0,Y 509.636,Z 266.664,A -85,B 0,C 180,E1 -5297.811,E2 -5297.811} C_VEL
LIN {X 0,Y 511.164,Z 276.69,A -85,B 0,C 180,E1 -5297.991,E2 -5297.991} C_VEL
LIN {X 0,Y 510.822,Z 341.841,A -85,B 0,C 180,E1 -5298.919,E2 -5298.919} C_VEL
LIN {X 0,Y 510.748,Z 351.008,A -85,B 0,C 180,E1 -5299.144,E2 -5299.144} C_VEL
LIN {X 0,Y 510.629,Z 359.419,A -85,B 0,C 180,E1 -5299.442,E2 -5299.442} C_VEL
LIN {X 0,Y 510.52,Z 366.938,A -85,B 0,C 180,E1 -5299.79,E2 -5299.79} C_VEL
LIN {X 0,Y 510.349,Z 375.408,A -85,B 0,C 180,E1 -5300.288,E2 -5300.288} C_VEL
LIN {X 0,Y 510.238,Z 383.531,A -85,B 0,C 180,E1 -5300.886,E2 -5300.886} C_VEL
LIN {X 0,Y 510.011,Z 391.243,A -85,B 0,C 180,E1 -5301.58,E2 -5301.58} C_VEL
LIN {X 0,Y 509.844,Z 397.605,A -85,B 0,C 180,E1 -5302.276,E2 -5302.276} C_VEL
LIN {X 0,Y 509.685,Z 404.985,A -85,B 0,C 180,E1 -5303.257,E2 -5303.257} C_VEL
LIN {X 0,Y 509.387,Z 411.927,A -85,B 0,C 180,E1 -5304.457,E2 -5304.457} C_VEL
LIN {X 0,Y 509.461,Z 415.581,A -85,B 0,C 180,E1 -5305.252,E2 -5305.252} C_VEL
LIN {X 0,Y 509.328,Z 418.57,A -85,B 0,C 180,E1 -5306.043,E2 -5306.043} C_VEL
LIN {X 0,Y 509.344,Z 420.88,A -85,B 0,C 180,E1 -5306.836,E2 -5306.836} C_VEL
LIN {X 0,Y 509.201,Z 422.652,A -85,B 0,C 180,E1 -5307.627,E2 -5307.627} C_VEL
LIN {X 0,Y 509.12,Z 423.929,A -85,B 0,C 180,E1 -5308.418,E2 -5308.418} C_VEL
LIN {X 0,Y 509.097,Z 424.737,A -85,B 0,C 180,E1 -5309.209,E2 -5309.209} C_VEL
LIN {X 0,Y 509.098,Z 425.044,A -85,B 0,C 180,E1 -5310,E2 -5310} C_VEL
LIN {X 0,Y 509.098,Z 424.774,A -85,B 0,C 180,E1 -5310.791,E2 -5310.791} C_VEL
LIN {X 0,Y 509.121,Z 424.039,A -85,B 0,C 180,E1 -5311.582,E2 -5311.582} C_VEL
LIN {X 0,Y 509.201,Z 422.837,A -85,B 0,C 180,E1 -5312.373,E2 -5312.373} C_VEL
LIN {X 0,Y 509.356,Z 420.003,A -85,B 0,C 180,E1 -5313.559,E2 -5313.559} C_VEL
LIN {X 0,Y 509.376,Z 417.432,A -85,B 0,C 180,E1 -5314.352,E2 -5314.352} C_VEL
LIN {X 0,Y 509.383,Z 412.364,A -85,B 0,C 180,E1 -5315.542,E2 -5315.542} C_VEL
LIN {X 0,Y 509.662,Z 406.598,A -85,B 0,C 180,E1 -5316.583,E2 -5316.583} C_VEL
LIN {X 0,Y 509.777,Z 400.041,A -85,B 0,C 180,E1 -5317.525,E2 -5317.525} C_VEL
LIN {X 0,Y 510.001,Z 391.146,A -85,B 0,C 180,E1 -5318.519,E2 -5318.519} C_VEL
LIN {X 0,Y 510.198,Z 384.64,A -85,B 0,C 180,E1 -5319.114,E2 -5319.114} C_VEL
LIN {X 0,Y 510.323,Z 376.763,A -85,B 0,C 180,E1 -5319.712,E2 -5319.712} C_VEL
LIN {X 0,Y 510.53,Z 368.626,A -85,B 0,C 180,E1 -5320.208,E2 -5320.208} C_VEL
LIN {X 0,Y 510.665,Z 360.392,A -85,B 0,C 180,E1 -5320.607,E2 -5320.607} C_VEL
LIN {X 0,Y 510.731,Z 351.521,A -85,B 0,C 180,E1 -5320.931,E2 -5320.931} C_VEL
LIN {X 0,Y 510.918,Z 342.874,A -85,B 0,C 180,E1 -5321.148,E2 -5321.148} C_VEL
LIN {X 0,Y 511.028,Z 290.717,A -85,B 0,C 180,E1 -5321.905,E2 -5321.905} C_VEL
LIN {X 0,Y 511.026,Z 274.981,A -85,B 0,C 180,E1 -5322.126,E2 -5322.126} C_VEL
LIN {X 0,Y 509.599,Z 266.343,A -85,B 0,C 180,E1 -5322.297,E2 -5322.297} C_VEL
LIN {X 0,Y 509.632,Z 253.362,A -85,B 0,C 180,E1 -5325.189,E2 -5325.189} C_VEL
LIN {X 0,Y 509.644,Z 251.821,A -85,B 0,C 180,E1 -5325.599,E2 -5325.599} C_VEL
LIN {X 0,Y 509.825,Z 251.791,A -85,B 0,C 180,E1 -5327.978,E2 -5327.978} C_VEL
LIN {X 0,Y 509.859,Z 251.784,A -85,B 0,C 180,E1 -5330.392,E2 -5330.392} C_VEL
LIN {X 0,Y 509.806,Z 251.795,A -85,B 0,C 180,E1 -5333.564,E2 -5333.564} C_VEL
LIN {X 0,Y 509.815,Z 251.79,A -85,B 0,C 180,E1 -5336.356,E2 -5336.356} C_VEL
LIN {X 0,Y 509.828,Z 251.792,A -85,B 0,C 180,E1 -5338.847,E2 -5338.847} C_VEL
LIN {X 0,Y 509.794,Z 251.796,A -85,B 0,C 180,E1 -5341.591,E2 -5341.591} C_VEL
LIN {X 0,Y 509.83,Z 251.789,A -85,B 0,C 180,E1 -5344.414,E2 -5344.414} C_VEL
LIN {X 0,Y 509.803,Z 251.796,A -85,B 0,C 180,E1 -5347.341,E2 -5347.341} C_VEL
LIN {X 0,Y 509.809,Z 251.792,A -85,B 0,C 180,E1 -5350.384,E2 -5350.384} C_VEL
LIN {X 0,Y 509.801,Z 251.793,A -85,B 0,C 180,E1 -5353.573,E2 -5353.573} C_VEL
LIN {X 0,Y 509.801,Z 251.795,A -85,B 0,C 180,E1 -5356.426,E2 -5356.426} C_VEL
LIN {X 0,Y 509.808,Z 251.791,A -85,B 0,C 180,E1 -5359.615,E2 -5359.615} C_VEL
LIN {X 0,Y 509.801,Z 251.796,A -85,B 0,C 180,E1 -5362.658,E2 -5362.658} C_VEL
LIN {X 0,Y 509.833,Z 251.788,A -85,B 0,C 180,E1 -5365.8,E2 -5365.8} C_VEL
LIN {X 0,Y 509.832,Z 251.793,A -85,B 0,C 180,E1 -5368.721,E2 -5368.721} C_VEL
LIN {X 0,Y 509.825,Z 251.79,A -85,B 0,C 180,E1 -5371.152,E2 -5371.152} C_VEL
LIN {X 0,Y 509.842,Z 251.788,A -85,B 0,C 180,E1 -5373.825,E2 -5373.825} C_VEL
LIN {X 0,Y 509.803,Z 251.796,A -85,B 0,C 180,E1 -5376.435,E2 -5376.435} C_VEL
LIN {X 0,Y 509.884,Z 251.784,A -85,B 0,C 180,E1 -5379.843,E2 -5379.843} C_VEL
LIN {X 0,Y 509.846,Z 251.791,A -85,B 0,C 180,E1 -5382.346,E2 -5382.346} C_VEL
LIN {X 0,Y 509.879,Z 251.784,A -85,B 0,C 180,E1 -5384.818,E2 -5384.818} C_VEL
LIN {X 0,Y 509.884,Z 251.786,A -85,B 0,C 180,E1 -5388.131,E2 -5388.131} C_VEL
LIN {X 0,Y 509.867,Z 251.784,A -85,B 0,C 180,E1 -5391.279,E2 -5391.279} C_VEL
LIN {X 0,Y 509.916,Z 251.781,A -85,B 0,C 180,E1 -5393.67,E2 -5393.67} C_VEL
LIN {X 0,Y 509.878,Z 251.782,A -85,B 0,C 180,E1 -5396.839,E2 -5396.839} C_VEL
LIN {X 0,Y 509.916,Z 251.78,A -85,B 0,C 180,E1 -5398.42,E2 -5398.42} C_VEL
LIN {X 0,Y 510.028,Z 251.769,A -85,B 0,C 180,E1 -5400,E2 -5400} C_VEL
LIN {X 0,Y 510.035,Z 251.765,A -85,B 0,C 180,E1 -5402.369,E2 -5402.369} C_VEL
LIN {X 0,Y 509.929,Z 251.779,A -85,B 0,C 180,E1 -5405.536,E2 -5405.536} C_VEL
LIN {X 0,Y 509.868,Z 251.79,A -85,B 0,C 180,E1 -5407.923,E2 -5407.923} C_VEL
LIN {X 0,Y 509.855,Z 251.786,A -85,B 0,C 180,E1 -5411.127,E2 -5411.127} C_VEL
LIN {X 0,Y 509.817,Z 251.794,A -85,B 0,C 180,E1 -5413.553,E2 -5413.553} C_VEL
LIN {X 0,Y 509.797,Z 251.795,A -85,B 0,C 180,E1 -5416.005,E2 -5416.005} C_VEL
LIN {X 0,Y 509.82,Z 251.789,A -85,B 0,C 180,E1 -5418.485,E2 -5418.485} C_VEL
LIN {X 0,Y 509.811,Z 251.792,A -85,B 0,C 180,E1 -5421.003,E2 -5421.003} C_VEL
LIN {X 0,Y 509.796,Z 251.799,A -85,B 0,C 180,E1 -5423.565,E2 -5423.565} C_VEL
LIN {X 0,Y 509.808,Z 251.79,A -85,B 0,C 180,E1 -5426.356,E2 -5426.356} C_VEL
LIN {X 0,Y 509.786,Z 251.795,A -85,B 0,C 180,E1 -5428.85,E2 -5428.85} C_VEL
LIN {X 0,Y 509.79,Z 251.796,A -85,B 0,C 180,E1 -5431.592,E2 -5431.592} C_VEL
LIN {X 0,Y 509.827,Z 251.788,A -85,B 0,C 180,E1 -5434.415,E2 -5434.415} C_VEL
LIN {X 0,Y 509.776,Z 251.8,A -85,B 0,C 180,E1 -5437.344,E2 -5437.344} C_VEL
LIN {X 0,Y 509.806,Z 251.791,A -85,B 0,C 180,E1 -5440.385,E2 -5440.385} C_VEL
LIN {X 0,Y 509.8,Z 251.792,A -85,B 0,C 180,E1 -5443.574,E2 -5443.574} C_VEL
LIN {X 0,Y 509.787,Z 251.794,A -85,B 0,C 180,E1 -5446.426,E2 -5446.426} C_VEL
LIN {X 0,Y 509.807,Z 251.79,A -85,B 0,C 180,E1 -5449.616,E2 -5449.616} C_VEL
LIN {X 0,Y 509.774,Z 251.799,A -85,B 0,C 180,E1 -5452.656,E2 -5452.656} C_VEL
LIN {X 0,Y 509.826,Z 251.787,A -85,B 0,C 180,E1 -5455.802,E2 -5455.802} C_VEL
LIN {X 0,Y 509.81,Z 251.797,A -85,B 0,C 180,E1 -5458.727,E2 -5458.727} C_VEL
LIN {X 0,Y 509.818,Z 251.791,A -85,B 0,C 180,E1 -5462.051,E2 -5462.051} C_VEL
LIN {X 0,Y 509.779,Z 251.801,A -85,B 0,C 180,E1 -5464.699,E2 -5464.699} C_VEL
LIN {X 0,Y 509.835,Z 251.909,A -85,B 0,C 180,E1 -5466.06,E2 -5466.06} C_VEL
LIN {X 0,Y 510.907,Z 258.992,A -85,B 0,C 180,E1 -5467.347,E2 -5467.347} C_VEL
LIN {X 0,Y 510.599,Z 273.592,A -85,B 0,C 180,E1 -5469.873,E2 -5469.873} C_VEL
LIN {X 0,Y 510.277,Z 289.352,A -85,B 0,C 180,E1 -5472.569,E2 -5472.569} C_VEL
LIN {X 0,Y 509.937,Z 308.674,A -85,B 0,C 180,E1 -5475.84,E2 -5475.84} C_VEL
LIN {X 0,Y 509.696,Z 319.961,A -85,B 0,C 180,E1 -5477.737,E2 -5477.737} C_VEL
LIN {X 0,Y 511.005,Z 332.875,A -85,B 0,C 180,E1 -5477.956,E2 -5477.956} C_VEL
LIN {X 0,Y 510.73,Z 398.254,A -85,B 0,C 180,E1 -5478.893,E2 -5478.893} C_VEL
LIN {X 0,Y 510.567,Z 408.732,A -85,B 0,C 180,E1 -5479.166,E2 -5479.166} C_VEL
LIN {X 0,Y 510.403,Z 419.464,A -85,B 0,C 180,E1 -5479.588,E2 -5479.588} C_VEL
LIN {X 0,Y 510.126,Z 430.116,A -85,B 0,C 180,E1 -5480.184,E2 -5480.184} C_VEL
LIN {X 0,Y 509.973,Z 438.467,A -85,B 0,C 180,E1 -5480.782,E2 -5480.782} C_VEL
LIN {X 0,Y 509.764,Z 446.371,A -85,B 0,C 180,E1 -5481.477,E2 -5481.477} C_VEL
LIN {X 0,Y 509.576,Z 453.765,A -85,B 0,C 180,E1 -5482.272,E2 -5482.272} C_VEL
LIN {X 0,Y 509.491,Z 460.255,A -85,B 0,C 180,E1 -5483.124,E2 -5483.124} C_VEL
LIN {X 0,Y 509.369,Z 467.167,A -85,B 0,C 180,E1 -5484.259,E2 -5484.259} C_VEL
LIN {X 0,Y 509.223,Z 471.805,A -85,B 0,C 180,E1 -5485.25,E2 -5485.25} C_VEL
LIN {X 0,Y 509.292,Z 474.828,A -85,B 0,C 180,E1 -5486.044,E2 -5486.044} C_VEL
LIN {X 0,Y 509.212,Z 477.164,A -85,B 0,C 180,E1 -5486.836,E2 -5486.836} C_VEL
LIN {X 0,Y 509.191,Z 478.925,A -85,B 0,C 180,E1 -5487.627,E2 -5487.627} C_VEL
LIN {X 0,Y 509.111,Z 480.182,A -85,B 0,C 180,E1 -5488.418,E2 -5488.418} C_VEL
LIN {X 0,Y 509.083,Z 480.966,A -85,B 0,C 180,E1 -5489.209,E2 -5489.209} C_VEL
LIN {X 0,Y 509.086,Z 481.263,A -85,B 0,C 180,E1 -5490,E2 -5490} C_VEL
LIN {X 0,Y 509.083,Z 480.966,A -85,B 0,C 180,E1 -5490.791,E2 -5490.791} C_VEL
LIN {X 0,Y 509.111,Z 480.18,A -85,B 0,C 180,E1 -5491.582,E2 -5491.582} C_VEL
LIN {X 0,Y 509.191,Z 478.922,A -85,B 0,C 180,E1 -5492.374,E2 -5492.374} C_VEL
LIN {X 0,Y 509.246,Z 476.001,A -85,B 0,C 180,E1 -5493.561,E2 -5493.561} C_VEL
LIN {X 0,Y 509.25,Z 473.336,A -85,B 0,C 180,E1 -5494.354,E2 -5494.354} C_VEL
LIN {X 0,Y 509.335,Z 468.125,A -85,B 0,C 180,E1 -5495.543,E2 -5495.543} C_VEL
LIN {X 0,Y 509.452,Z 461.766,A -85,B 0,C 180,E1 -5496.659,E2 -5496.659} C_VEL
LIN {X 0,Y 509.577,Z 453.76,A -85,B 0,C 180,E1 -5497.728,E2 -5497.728} C_VEL
LIN {X 0,Y 509.765,Z 446.369,A -85,B 0,C 180,E1 -5498.523,E2 -5498.523} C_VEL
LIN {X 0,Y 509.974,Z 438.46,A -85,B 0,C 180,E1 -5499.219,E2 -5499.219} C_VEL
LIN {X 0,Y 510.127,Z 430.105,A -85,B 0,C 180,E1 -5499.817,E2 -5499.817} C_VEL
LIN {X 0,Y 510.404,Z 419.451,A -85,B 0,C 180,E1 -5500.412,E2 -5500.412} C_VEL
LIN {X 0,Y 510.557,Z 407.874,A -85,B 0,C 180,E1 -5500.861,E2 -5500.861} C_VEL
LIN {X 0,Y 510.741,Z 398.213,A -85,B 0,C 180,E1 -5501.108,E2 -5501.108} C_VEL
LIN {X 0,Y 511.004,Z 331.83,A -85,B 0,C 180,E1 -5502.058,E2 -5502.058} C_VEL
LIN {X 0,Y 509.714,Z 319.921,A -85,B 0,C 180,E1 -5502.27,E2 -5502.27} C_VEL
LIN {X 0,Y 509.949,Z 303.845,A -85,B 0,C 180,E1 -5504.976,E2 -5504.976} C_VEL
LIN {X 0,Y 510.468,Z 283.296,A -85,B 0,C 180,E1 -5508.461,E2 -5508.461} C_VEL
LIN {X 0,Y 510.815,Z 263.858,A -85,B 0,C 180,E1 -5511.807,E2 -5511.807} C_VEL
LIN {X 0,Y 510.875,Z 258.024,A -85,B 0,C 180,E1 -5512.824,E2 -5512.824} C_VEL
LIN {X 0,Y 509.848,Z 251.789,A -85,B 0,C 180,E1 -5513.994,E2 -5513.994} C_VEL
LIN {X 0,Y 509.813,Z 251.795,A -85,B 0,C 180,E1 -5517.06,E2 -5517.06} C_VEL
LIN {X 0,Y 509.783,Z 251.795,A -85,B 0,C 180,E1 -5519.756,E2 -5519.756} C_VEL
LIN {X 0,Y 509.821,Z 251.79,A -85,B 0,C 180,E1 -5522.765,E2 -5522.765} C_VEL
LIN {X 0,Y 509.777,Z 251.797,A -85,B 0,C 180,E1 -5525.571,E2 -5525.571} C_VEL
LIN {X 0,Y 509.801,Z 251.79,A -85,B 0,C 180,E1 -5528.343,E2 -5528.343} C_VEL
LIN {X 0,Y 509.784,Z 251.796,A -85,B 0,C 180,E1 -5531.433,E2 -5531.433} C_VEL
LIN {X 0,Y 509.835,Z 251.79,A -85,B 0,C 180,E1 -5534.671,E2 -5534.671} C_VEL
LIN {X 0,Y 509.787,Z 251.794,A -85,B 0,C 180,E1 -5537.505,E2 -5537.505} C_VEL
LIN {X 0,Y 509.822,Z 251.793,A -85,B 0,C 180,E1 -5540.645,E2 -5540.645} C_VEL
LIN {X 0,Y 509.763,Z 251.796,A -85,B 0,C 180,E1 -5543.642,E2 -5543.642} C_VEL
LIN {X 0,Y 509.824,Z 251.793,A -85,B 0,C 180,E1 -5546.537,E2 -5546.537} C_VEL
LIN {X 0,Y 509.801,Z 251.793,A -85,B 0,C 180,E1 -5549.331,E2 -5549.331} C_VEL
LIN {X 0,Y 509.822,Z 251.79,A -85,B 0,C 180,E1 -5552.05,E2 -5552.05} C_VEL
LIN {X 0,Y 509.783,Z 251.799,A -85,B 0,C 180,E1 -5554.699,E2 -5554.699} C_VEL
LIN {X 0,Y 509.824,Z 251.788,A -85,B 0,C 180,E1 -5557.459,E2 -5557.459} C_VEL
LIN {X 0,Y 509.807,Z 251.795,A -85,B 0,C 180,E1 -5560.679,E2 -5560.679} C_VEL
LIN {X 0,Y 509.788,Z 251.794,A -85,B 0,C 180,E1 -5563.172,E2 -5563.172} C_VEL
LIN {X 0,Y 509.814,Z 251.79,A -85,B 0,C 180,E1 -5565.633,E2 -5565.633} C_VEL
LIN {X 0,Y 509.889,Z 251.786,A -85,B 0,C 180,E1 -5568.132,E2 -5568.132} C_VEL
LIN {X 0,Y 509.872,Z 251.783,A -85,B 0,C 180,E1 -5571.279,E2 -5571.279} C_VEL
LIN {X 0,Y 509.916,Z 251.779,A -85,B 0,C 180,E1 -5573.67,E2 -5573.67} C_VEL
LIN {X 0,Y 509.883,Z 251.782,A -85,B 0,C 180,E1 -5576.84,E2 -5576.84} C_VEL
LIN {X 0,Y 509.923,Z 251.78,A -85,B 0,C 180,E1 -5578.421,E2 -5578.421} C_VEL
LIN {X 0,Y 510.034,Z 251.768,A -85,B 0,C 180,E1 -5580,E2 -5580} C_VEL
LIN {X 0,Y 510.041,Z 251.766,A -85,B 0,C 180,E1 -5582.369,E2 -5582.369} C_VEL
LIN {X 0,Y 509.935,Z 251.778,A -85,B 0,C 180,E1 -5585.536,E2 -5585.536} C_VEL
LIN {X 0,Y 509.875,Z 251.787,A -85,B 0,C 180,E1 -5587.923,E2 -5587.923} C_VEL
LIN {X 0,Y 509.862,Z 251.785,A -85,B 0,C 180,E1 -5591.127,E2 -5591.127} C_VEL
LIN {X 0,Y 509.824,Z 251.794,A -85,B 0,C 180,E1 -5593.553,E2 -5593.553} C_VEL
LIN {X 0,Y 509.805,Z 251.796,A -85,B 0,C 180,E1 -5596.005,E2 -5596.005} C_VEL
LIN {X 0,Y 509.827,Z 251.789,A -85,B 0,C 180,E1 -5598.485,E2 -5598.485} C_VEL
LIN {X 0,Y 509.818,Z 251.791,A -85,B 0,C 180,E1 -5601.003,E2 -5601.003} C_VEL
LIN {X 0,Y 509.809,Z 251.795,A -85,B 0,C 180,E1 -5603.565,E2 -5603.565} C_VEL
LIN {X 0,Y 509.816,Z 251.79,A -85,B 0,C 180,E1 -5606.356,E2 -5606.356} C_VEL
LIN {X 0,Y 509.824,Z 251.79,A -85,B 0,C 180,E1 -5608.848,E2 -5608.848} C_VEL
LIN {X 0,Y 509.812,Z 251.795,A -85,B 0,C 180,E1 -5611.591,E2 -5611.591} C_VEL
LIN {X 0,Y 509.834,Z 251.788,A -85,B 0,C 180,E1 -5614.415,E2 -5614.415} C_VEL
LIN {X 0,Y 509.807,Z 251.795,A -85,B 0,C 180,E1 -5617.342,E2 -5617.342} C_VEL
LIN {X 0,Y 509.813,Z 251.79,A -85,B 0,C 180,E1 -5620.385,E2 -5620.385} C_VEL
LIN {X 0,Y 509.806,Z 251.795,A -85,B 0,C 180,E1 -5623.573,E2 -5623.573} C_VEL
LIN {X 0,Y 509.806,Z 251.792,A -85,B 0,C 180,E1 -5626.426,E2 -5626.426} C_VEL
LIN {X 0,Y 509.814,Z 251.792,A -85,B 0,C 180,E1 -5629.615,E2 -5629.615} C_VEL
LIN {X 0,Y 509.809,Z 251.794,A -85,B 0,C 180,E1 -5632.658,E2 -5632.658} C_VEL
LIN {X 0,Y 509.808,Z 251.792,A -85,B 0,C 180,E1 -5633.692,E2 -5633.692} C_VEL
LIN {X 0,Y 509.141,Z 251.876,A -85,B 0,C 180,E1 -5634.352,E2 -5634.352} C_VEL
LIN {X 0,Y 506.321,Z 252.229,A -85,B 0,C 180,E1 -5635.424,E2 -5635.424} C_VEL
LIN {X 0,Y 503.929,Z 252.53,A -85,B 0,C 180,E1 -5636.287,E2 -5636.287} C_VEL
LIN {X 0,Y 502.884,Z 252.658,A -85,B 0,C 180,E1 -5636.954,E2 -5636.954} C_VEL
LIN {X 0,Y 502.788,Z 252.668,A -85,B 0,C 180,E1 -5637.179,E2 -5637.179} C_VEL
LIN {X 0,Y 502.791,Z 252.665,A -85,B 0,C 180,E1 -5640.07,E2 -5640.07} C_VEL
LIN {X 0,Y 502.778,Z 252.67,A -85,B 0,C 180,E1 -5642.53,E2 -5642.53} C_VEL
LIN {X 0,Y 502.772,Z 252.669,A -85,B 0,C 180,E1 -5645.313,E2 -5645.313} C_VEL
LIN {X 0,Y 502.778,Z 252.667,A -85,B 0,C 180,E1 -5647.826,E2 -5647.826} C_VEL
LIN {X 0,Y 502.811,Z 252.668,A -85,B 0,C 180,E1 -5650.399,E2 -5650.399} C_VEL
LIN {X 0,Y 502.754,Z 252.675,A -85,B 0,C 180,E1 -5652.929,E2 -5652.929} C_VEL
LIN {X 0,Y 502.609,Z 252.791,A -85,B 0,C 180,E1 -5654.54,E2 -5654.54} C_VEL
LIN {X 0,Y 502.574,Z 266.681,A -85,B 0,C 180,E1 -5657.631,E2 -5657.631} C_VEL
LIN {X 0,Y 504.223,Z 276.473,A -85,B 0,C 180,E1 -5657.814,E2 -5657.814} C_VEL
LIN {X 0,Y 503.879,Z 342.264,A -85,B 0,C 180,E1 -5658.765,E2 -5658.765} C_VEL
LIN {X 0,Y 503.791,Z 351.42,A -85,B 0,C 180,E1 -5658.992,E2 -5658.992} C_VEL
LIN {X 0,Y 503.685,Z 359.824,A -85,B 0,C 180,E1 -5659.295,E2 -5659.295} C_VEL
LIN {X 0,Y 503.566,Z 367.34,A -85,B 0,C 180,E1 -5659.648,E2 -5659.648} C_VEL
LIN {X 0,Y 503.361,Z 375.809,A -85,B 0,C 180,E1 -5660.152,E2 -5660.152} C_VEL
LIN {X 0,Y 503.253,Z 383.929,A -85,B 0,C 180,E1 -5660.758,E2 -5660.758} C_VEL
LIN {X 0,Y 503.004,Z 391.641,A -85,B 0,C 180,E1 -5661.462,E2 -5661.462} C_VEL
LIN {X 0,Y 502.815,Z 398.002,A -85,B 0,C 180,E1 -5662.167,E2 -5662.167} C_VEL
LIN {X 0,Y 502.66,Z 404.741,A -85,B 0,C 180,E1 -5663.071,E2 -5663.071} C_VEL
LIN {X 0,Y 502.415,Z 411.358,A -85,B 0,C 180,E1 -5664.179,E2 -5664.179} C_VEL
LIN {X 0,Y 502.411,Z 415.974,A -85,B 0,C 180,E1 -5665.185,E2 -5665.185} C_VEL
LIN {X 0,Y 502.269,Z 418.963,A -85,B 0,C 180,E1 -5665.988,E2 -5665.988} C_VEL
LIN {X 0,Y 502.287,Z 421.272,A -85,B 0,C 180,E1 -5666.791,E2 -5666.791} C_VEL
LIN {X 0,Y 502.136,Z 423.043,A -85,B 0,C 180,E1 -5667.593,E2 -5667.593} C_VEL
LIN {X 0,Y 502.044,Z 424.321,A -85,B 0,C 180,E1 -5668.395,E2 -5668.395} C_VEL
LIN {X 0,Y 502.013,Z 425.129,A -85,B 0,C 180,E1 -5669.197,E2 -5669.197} C_VEL
LIN {X 0,Y 502.011,Z 425.436,A -85,B 0,C 180,E1 -5670,E2 -5670} C_VEL
LIN {X 0,Y 502.013,Z 425.165,A -85,B 0,C 180,E1 -5670.802,E2 -5670.802} C_VEL
LIN {X 0,Y 502.044,Z 424.429,A -85,B 0,C 180,E1 -5671.604,E2 -5671.604} C_VEL
LIN {X 0,Y 502.136,Z 423.226,A -85,B 0,C 180,E1 -5672.406,E2 -5672.406} C_VEL
LIN {X 0,Y 502.297,Z 420.392,A -85,B 0,C 180,E1 -5673.609,E2 -5673.609} C_VEL
LIN {X 0,Y 502.322,Z 417.82,A -85,B 0,C 180,E1 -5674.413,E2 -5674.413} C_VEL
LIN {X 0,Y 502.337,Z 412.751,A -85,B 0,C 180,E1 -5675.62,E2 -5675.62} C_VEL
LIN {X 0,Y 502.622,Z 407.319,A -85,B 0,C 180,E1 -5676.617,E2 -5676.617} C_VEL
LIN {X 0,Y 502.747,Z 400.428,A -85,B 0,C 180,E1 -5677.631,E2 -5677.631} C_VEL
LIN {X 0,Y 503.002,Z 392.544,A -85,B 0,C 180,E1 -5678.537,E2 -5678.537} C_VEL
LIN {X 0,Y 503.216,Z 385.023,A -85,B 0,C 180,E1 -5679.242,E2 -5679.242} C_VEL
LIN {X 0,Y 503.349,Z 377.144,A -85,B 0,C 180,E1 -5679.848,E2 -5679.848} C_VEL
LIN {X 0,Y 503.553,Z 369.005,A -85,B 0,C 180,E1 -5680.351,E2 -5680.351} C_VEL
LIN {X 0,Y 503.697,Z 360.769,A -85,B 0,C 180,E1 -5680.755,E2 -5680.755} C_VEL
LIN {X 0,Y 503.782,Z 351.891,A -85,B 0,C 180,E1 -5681.084,E2 -5681.084} C_VEL
LIN {X 0,Y 503.946,Z 343.328,A -85,B 0,C 180,E1 -5681.303,E2 -5681.303} C_VEL
LIN {X 0,Y 504.184,Z 279.258,A -85,B 0,C 180,E1 -5682.237,E2 -5682.237} C_VEL
LIN {X 0,Y 503.911,Z 274.542,A -85,B 0,C 180,E1 -5682.312,E2 -5682.312} C_VEL
LIN {X 0,Y 502.579,Z 266.643,A -85,B 0,C 180,E1 -5682.466,E2 -5682.466} C_VEL
LIN {X 0,Y 502.581,Z 252.965,A -85,B 0,C 180,E1 -5685.512,E2 -5685.512} C_VEL
LIN {X 0,Y 502.666,Z 252.689,A -85,B 0,C 180,E1 -5685.821,E2 -5685.821} C_VEL
LIN {X 0,Y 502.805,Z 252.664,A -85,B 0,C 180,E1 -5688.752,E2 -5688.752} C_VEL
LIN {X 0,Y 502.768,Z 252.673,A -85,B 0,C 180,E1 -5691.311,E2 -5691.311} C_VEL
LIN {X 0,Y 502.758,Z 252.671,A -85,B 0,C 180,E1 -5693.915,E2 -5693.915} C_VEL
LIN {X 0,Y 502.782,Z 252.667,A -85,B 0,C 180,E1 -5696.57,E2 -5696.57} C_VEL
LIN {X 0,Y 502.787,Z 252.666,A -85,B 0,C 180,E1 -5699.929,E2 -5699.929} C_VEL
LIN {X 0,Y 502.8,Z 252.669,A -85,B 0,C 180,E1 -5703.033,E2 -5703.033} C_VEL
LIN {X 0,Y 502.759,Z 252.669,A -85,B 0,C 180,E1 -5705.952,E2 -5705.952} C_VEL
LIN {X 0,Y 502.789,Z 252.67,A -85,B 0,C 180,E1 -5708.976,E2 -5708.976} C_VEL
LIN {X 0,Y 502.741,Z 252.672,A -85,B 0,C 180,E1 -5712.191,E2 -5712.191} C_VEL
LIN {X 0,Y 502.782,Z 252.668,A -85,B 0,C 180,E1 -5715.47,E2 -5715.47} C_VEL
LIN {X 0,Y 502.757,Z 252.673,A -85,B 0,C 180,E1 -5718.928,E2 -5718.928} C_VEL
LIN {X 0,Y 502.767,Z 252.669,A -85,B 0,C 180,E1 -5722.044,E2 -5722.044} C_VEL
LIN {X 0,Y 502.783,Z 252.67,A -85,B 0,C 180,E1 -5725.033,E2 -5725.033} C_VEL
LIN {X 0,Y 502.773,Z 252.668,A -85,B 0,C 180,E1 -5727.915,E2 -5727.915} C_VEL
LIN {X 0,Y 502.784,Z 252.67,A -85,B 0,C 180,E1 -5730.71,E2 -5730.71} C_VEL
LIN {X 0,Y 502.768,Z 252.668,A -85,B 0,C 180,E1 -5733.46,E2 -5733.46} C_VEL
LIN {X 0,Y 502.755,Z 252.674,A -85,B 0,C 180,E1 -5736.084,E2 -5736.084} C_VEL
LIN {X 0,Y 502.825,Z 252.661,A -85,B 0,C 180,E1 -5739.464,E2 -5739.464} C_VEL
LIN {X 0,Y 502.794,Z 252.669,A -85,B 0,C 180,E1 -5742.09,E2 -5742.09} C_VEL
LIN {X 0,Y 502.818,Z 252.662,A -85,B 0,C 180,E1 -5745.428,E2 -5745.428} C_VEL
LIN {X 0,Y 502.831,Z 252.662,A -85,B 0,C 180,E1 -5748.716,E2 -5748.716} C_VEL
LIN {X 0,Y 502.84,Z 252.663,A -85,B 0,C 180,E1 -5751.966,E2 -5751.966} C_VEL
LIN {X 0,Y 502.89,Z 252.657,A -85,B 0,C 180,E1 -5754.386,E2 -5754.386} C_VEL
LIN {X 0,Y 503.003,Z 252.642,A -85,B 0,C 180,E1 -5757.598,E2 -5757.598} C_VEL
LIN {X 0,Y 502.997,Z 252.644,A -85,B 0,C 180,E1 -5760,E2 -5760} C_VEL
LIN {X 0,Y 503.002,Z 252.641,A -85,B 0,C 180,E1 -5762.402,E2 -5762.402} C_VEL
LIN {X 0,Y 502.886,Z 252.657,A -85,B 0,C 180,E1 -5765.614,E2 -5765.614} C_VEL
LIN {X 0,Y 502.84,Z 252.664,A -85,B 0,C 180,E1 -5768.034,E2 -5768.034} C_VEL
LIN {X 0,Y 502.83,Z 252.663,A -85,B 0,C 180,E1 -5771.284,E2 -5771.284} C_VEL
LIN {X 0,Y 502.817,Z 252.661,A -85,B 0,C 180,E1 -5774.572,E2 -5774.572} C_VEL
LIN {X 0,Y 502.778,Z 252.67,A -85,B 0,C 180,E1 -5777.91,E2 -5777.91} C_VEL
LIN {X 0,Y 502.796,Z 252.664,A -85,B 0,C 180,E1 -5780.528,E2 -5780.528} C_VEL
LIN {X 0,Y 502.773,Z 252.67,A -85,B 0,C 180,E1 -5783.041,E2 -5783.041} C_VEL
LIN {X 0,Y 502.769,Z 252.672,A -85,B 0,C 180,E1 -5785.679,E2 -5785.679} C_VEL
LIN {X 0,Y 502.753,Z 252.669,A -85,B 0,C 180,E1 -5788.378,E2 -5788.378} C_VEL
LIN {X 0,Y 502.764,Z 252.673,A -85,B 0,C 180,E1 -5791.494,E2 -5791.494} C_VEL
LIN {X 0,Y 502.779,Z 252.666,A -85,B 0,C 180,E1 -5794.441,E2 -5794.441} C_VEL
LIN {X 0,Y 502.731,Z 252.678,A -85,B 0,C 180,E1 -5797.172,E2 -5797.172} C_VEL
LIN {X 0,Y 502.763,Z 252.667,A -85,B 0,C 180,E1 -5800.017,E2 -5800.017} C_VEL
LIN {X 0,Y 502.741,Z 252.676,A -85,B 0,C 180,E1 -5803.235,E2 -5803.235} C_VEL
LIN {X 0,Y 502.762,Z 252.668,A -85,B 0,C 180,E1 -5805.659,E2 -5805.659} C_VEL
LIN {X 0,Y 502.758,Z 252.675,A -85,B 0,C 180,E1 -5809.013,E2 -5809.013} C_VEL
LIN {X 0,Y 502.754,Z 252.669,A -85,B 0,C 180,E1 -5812.043,E2 -5812.043} C_VEL
LIN {X 0,Y 502.775,Z 252.67,A -85,B 0,C 180,E1 -5815.033,E2 -5815.033} C_VEL
LIN {X 0,Y 502.751,Z 252.669,A -85,B 0,C 180,E1 -5817.914,E2 -5817.914} C_VEL
LIN {X 0,Y 502.748,Z 252.677,A -85,B 0,C 180,E1 -5820.708,E2 -5820.708} C_VEL
LIN {X 0,Y 502.766,Z 252.669,A -85,B 0,C 180,E1 -5823.461,E2 -5823.461} C_VEL
LIN {X 0,Y 502.8,Z 252.737,A -85,B 0,C 180,E1 -5825.923,E2 -5825.923} C_VEL
LIN {X 0,Y 503.911,Z 259.305,A -85,B 0,C 180,E1 -5827.139,E2 -5827.139} C_VEL
LIN {X 0,Y 503.583,Z 274.42,A -85,B 0,C 180,E1 -5829.794,E2 -5829.794} C_VEL
LIN {X 0,Y 503.266,Z 288.968,A -85,B 0,C 180,E1 -5832.319,E2 -5832.319} C_VEL
LIN {X 0,Y 502.904,Z 308.289,A -85,B 0,C 180,E1 -5835.638,E2 -5835.638} C_VEL
LIN {X 0,Y 502.642,Z 319.521,A -85,B 0,C 180,E1 -5837.553,E2 -5837.553} C_VEL
LIN {X 0,Y 504.076,Z 333.667,A -85,B 0,C 180,E1 -5837.805,E2 -5837.805} C_VEL
LIN {X 0,Y 503.773,Z 397.862,A -85,B 0,C 180,E1 -5838.738,E2 -5838.738} C_VEL
LIN {X 0,Y 503.564,Z 408.339,A -85,B 0,C 180,E1 -5839.013,E2 -5839.013} C_VEL
LIN {X 0,Y 503.408,Z 419.071,A -85,B 0,C 180,E1 -5839.442,E2 -5839.442} C_VEL
LIN {X 0,Y 503.124,Z 429.724,A -85,B 0,C 180,E1 -5840.046,E2 -5840.046} C_VEL
LIN {X 0,Y 502.959,Z 438.075,A -85,B 0,C 180,E1 -5840.652,E2 -5840.652} C_VEL
LIN {X 0,Y 502.694,Z 445.976,A -85,B 0,C 180,E1 -5841.357,E2 -5841.357} C_VEL
LIN {X 0,Y 502.515,Z 453.371,A -85,B 0,C 180,E1 -5842.163,E2 -5842.163} C_VEL
LIN {X 0,Y 502.368,Z 461.149,A -85,B 0,C 180,E1 -5843.211,E2 -5843.211} C_VEL
LIN {X 0,Y 502.259,Z 467.739,A -85,B 0,C 180,E1 -5844.379,E2 -5844.379} C_VEL
LIN {X 0,Y 502.145,Z 472.946,A -85,B 0,C 180,E1 -5845.586,E2 -5845.586} C_VEL
LIN {X 0,Y 502.17,Z 475.612,A -85,B 0,C 180,E1 -5846.39,E2 -5846.39} C_VEL
LIN {X 0,Y 502.122,Z 478.534,A -85,B 0,C 180,E1 -5847.594,E2 -5847.594} C_VEL
LIN {X 0,Y 502.035,Z 479.791,A -85,B 0,C 180,E1 -5848.396,E2 -5848.396} C_VEL
LIN {X 0,Y 501.999,Z 480.575,A -85,B 0,C 180,E1 -5849.198,E2 -5849.198} C_VEL
LIN {X 0,Y 502,Z 480.872,A -85,B 0,C 180,E1 -5850,E2 -5850} C_VEL
LIN {X 0,Y 501.999,Z 480.574,A -85,B 0,C 180,E1 -5850.803,E2 -5850.803} C_VEL
LIN {X 0,Y 502.035,Z 479.79,A -85,B 0,C 180,E1 -5851.605,E2 -5851.605} C_VEL
LIN {X 0,Y 502.122,Z 478.531,A -85,B 0,C 180,E1 -5852.407,E2 -5852.407} C_VEL
LIN {X 0,Y 502.17,Z 475.609,A -85,B 0,C 180,E1 -5853.611,E2 -5853.611} C_VEL
LIN {X 0,Y 502.146,Z 472.942,A -85,B 0,C 180,E1 -5854.415,E2 -5854.415} C_VEL
LIN {X 0,Y 502.259,Z 467.732,A -85,B 0,C 180,E1 -5855.621,E2 -5855.621} C_VEL
LIN {X 0,Y 502.366,Z 462.007,A -85,B 0,C 180,E1 -5856.649,E2 -5856.649} C_VEL
LIN {X 0,Y 502.475,Z 455.074,A -85,B 0,C 180,E1 -5857.636,E2 -5857.636} C_VEL
LIN {X 0,Y 502.673,Z 447.002,A -85,B 0,C 180,E1 -5858.543,E2 -5858.543} C_VEL
LIN {X 0,Y 502.91,Z 439.303,A -85,B 0,C 180,E1 -5859.248,E2 -5859.248} C_VEL
LIN {X 0,Y 503.082,Z 431.219,A -85,B 0,C 180,E1 -5859.854,E2 -5859.854} C_VEL
LIN {X 0,Y 503.274,Z 422.85,A -85,B 0,C 180,E1 -5860.358,E2 -5860.358} C_VEL
LIN {X 0,Y 503.475,Z 414.316,A -85,B 0,C 180,E1 -5860.761,E2 -5860.761} C_VEL
LIN {X 0,Y 503.668,Z 404.985,A -85,B 0,C 180,E1 -5861.087,E2 -5861.087} C_VEL
LIN {X 0,Y 503.802,Z 394.418,A -85,B 0,C 180,E1 -5861.329,E2 -5861.329} C_VEL
LIN {X 0,Y 503.941,Z 331.432,A -85,B 0,C 180,E1 -5862.23,E2 -5862.23} C_VEL
LIN {X 0,Y 502.647,Z 319.616,A -85,B 0,C 180,E1 -5862.431,E2 -5862.431} C_VEL
LIN {X 0,Y 502.903,Z 304.752,A -85,B 0,C 180,E1 -5864.968,E2 -5864.968} C_VEL
LIN {X 0,Y 503.374,Z 285.357,A -85,B 0,C 180,E1 -5868.305,E2 -5868.305} C_VEL
LIN {X 0,Y 503.733,Z 267.119,A -85,B 0,C 180,E1 -5871.484,E2 -5871.484} C_VEL
LIN {X 0,Y 503.796,Z 258.585,A -85,B 0,C 180,E1 -5872.992,E2 -5872.992} C_VEL
LIN {X 0,Y 502.809,Z 252.665,A -85,B 0,C 180,E1 -5874.132,E2 -5874.132} C_VEL
LIN {X 0,Y 502.768,Z 252.674,A -85,B 0,C 180,E1 -5877.471,E2 -5877.471} C_VEL
LIN {X 0,Y 502.742,Z 252.669,A -85,B 0,C 180,E1 -5880.216,E2 -5880.216} C_VEL
LIN {X 0,Y 502.768,Z 252.671,A -85,B 0,C 180,E1 -5883.036,E2 -5883.036} C_VEL
LIN {X 0,Y 502.737,Z 252.671,A -85,B 0,C 180,E1 -5885.955,E2 -5885.955} C_VEL
LIN {X 0,Y 502.766,Z 252.673,A -85,B 0,C 180,E1 -5888.98,E2 -5888.98} C_VEL
LIN {X 0,Y 502.745,Z 252.67,A -85,B 0,C 180,E1 -5892.192,E2 -5892.192} C_VEL
LIN {X 0,Y 502.778,Z 252.668,A -85,B 0,C 180,E1 -5895.471,E2 -5895.471} C_VEL
LIN {X 0,Y 502.757,Z 252.675,A -85,B 0,C 180,E1 -5898.928,E2 -5898.928} C_VEL
LIN {X 0,Y 502.753,Z 252.669,A -85,B 0,C 180,E1 -5902.043,E2 -5902.043} C_VEL
LIN {X 0,Y 502.776,Z 252.67,A -85,B 0,C 180,E1 -5905.032,E2 -5905.032} C_VEL
LIN {X 0,Y 502.755,Z 252.669,A -85,B 0,C 180,E1 -5907.913,E2 -5907.913} C_VEL
LIN {X 0,Y 502.752,Z 252.675,A -85,B 0,C 180,E1 -5910.708,E2 -5910.708} C_VEL
LIN {X 0,Y 502.77,Z 252.667,A -85,B 0,C 180,E1 -5913.461,E2 -5913.461} C_VEL
LIN {X 0,Y 502.746,Z 252.672,A -85,B 0,C 180,E1 -5916.084,E2 -5916.084} C_VEL
LIN {X 0,Y 502.755,Z 252.673,A -85,B 0,C 180,E1 -5918.688,E2 -5918.688} C_VEL
LIN {X 0,Y 502.787,Z 252.667,A -85,B 0,C 180,E1 -5921.899,E2 -5921.899} C_VEL
LIN {X 0,Y 502.792,Z 252.668,A -85,B 0,C 180,E1 -5924.683,E2 -5924.683} C_VEL
LIN {X 0,Y 502.84,Z 252.663,A -85,B 0,C 180,E1 -5928.06,E2 -5928.06} C_VEL
LIN {X 0,Y 502.836,Z 252.659,A -85,B 0,C 180,E1 -5931.156,E2 -5931.156} C_VEL
LIN {X 0,Y 502.866,Z 252.657,A -85,B 0,C 180,E1 -5933.581,E2 -5933.581} C_VEL
LIN {X 0,Y 502.829,Z 252.662,A -85,B 0,C 180,E1 -5936.795,E2 -5936.795} C_VEL
LIN {X 0,Y 502.893,Z 252.656,A -85,B 0,C 180,E1 -5938.398,E2 -5938.398} C_VEL
LIN {X 0,Y 503.003,Z 252.644,A -85,B 0,C 180,E1 -5940,E2 -5940} C_VEL
LIN {X 0,Y 503.008,Z 252.641,A -85,B 0,C 180,E1 -5942.402,E2 -5942.402} C_VEL
LIN {X 0,Y 502.892,Z 252.656,A -85,B 0,C 180,E1 -5945.614,E2 -5945.614} C_VEL
LIN {X 0,Y 502.847,Z 252.662,A -85,B 0,C 180,E1 -5948.034,E2 -5948.034} C_VEL
LIN {X 0,Y 502.838,Z 252.661,A -85,B 0,C 180,E1 -5951.284,E2 -5951.284} C_VEL
LIN {X 0,Y 502.825,Z 252.662,A -85,B 0,C 180,E1 -5954.572,E2 -5954.572} C_VEL
LIN {X 0,Y 502.785,Z 252.67,A -85,B 0,C 180,E1 -5957.91,E2 -5957.91} C_VEL
LIN {X 0,Y 502.803,Z 252.664,A -85,B 0,C 180,E1 -5960.528,E2 -5960.528} C_VEL
LIN {X 0,Y 502.782,Z 252.668,A -85,B 0,C 180,E1 -5963.041,E2 -5963.041} C_VEL
LIN {X 0,Y 502.777,Z 252.671,A -85,B 0,C 180,E1 -5965.679,E2 -5965.679} C_VEL
LIN {X 0,Y 502.768,Z 252.668,A -85,B 0,C 180,E1 -5968.377,E2 -5968.377} C_VEL
LIN {X 0,Y 502.785,Z 252.67,A -85,B 0,C 180,E1 -5971.144,E2 -5971.144} C_VEL
LIN {X 0,Y 502.787,Z 252.668,A -85,B 0,C 180,E1 -5973.995,E2 -5973.995} C_VEL
LIN {X 0,Y 502.763,Z 252.673,A -85,B 0,C 180,E1 -5977.175,E2 -5977.175} C_VEL
LIN {X 0,Y 502.771,Z 252.669,A -85,B 0,C 180,E1 -5980.017,E2 -5980.017} C_VEL
LIN {X 0,Y 502.747,Z 252.675,A -85,B 0,C 180,E1 -5983.234,E2 -5983.234} C_VEL
LIN {X 0,Y 502.78,Z 252.669,A -85,B 0,C 180,E1 -5985.66,E2 -5985.66} C_VEL
LIN {X 0,Y 502.765,Z 252.672,A -85,B 0,C 180,E1 -5989.012,E2 -5989.012} C_VEL
LIN {X 0,Y 502.791,Z 252.665,A -85,B 0,C 180,E1 -5992.046,E2 -5992.046} C_VEL
LIN {X 0,Y 502.793,Z 252.669,A -85,B 0,C 180,E1 -5995.033,E2 -5995.033} C_VEL
LIN {X 0,Y 502.788,Z 252.668,A -85,B 0,C 180,E1 -5997.179,E2 -5997.179} C_VEL
LIN {X 0,Y 502.093,Z 252.753,A -85,B 0,C 180,E1 -5997.848,E2 -5997.848} C_VEL
LIN {X 0,Y 499.233,Z 253.113,A -85,B 0,C 180,E1 -5998.934,E2 -5998.934} C_VEL
LIN {X 0,Y 496.831,Z 253.41,A -85,B 0,C 180,E1 -5999.809,E2 -5999.809} C_VEL
LIN {X 0,Y 495.8,Z 253.54,A -85,B 0,C 180,E1 -6000.484,E2 -6000.484} C_VEL
LIN {X 0,Y 495.715,Z 253.547,A -85,B 0,C 180,E1 -6000.713,E2 -6000.713} C_VEL
LIN {X 0,Y 495.719,Z 253.546,A -85,B 0,C 180,E1 -6003.928,E2 -6003.928} C_VEL
LIN {X 0,Y 495.747,Z 253.546,A -85,B 0,C 180,E1 -6007.143,E2 -6007.143} C_VEL
LIN {X 0,Y 495.761,Z 253.543,A -85,B 0,C 180,E1 -6010.109,E2 -6010.109} C_VEL
LIN {X 0,Y 495.713,Z 253.553,A -85,B 0,C 180,E1 -6012.678,E2 -6012.678} C_VEL
LIN {X 0,Y 495.576,Z 253.63,A -85,B 0,C 180,E1 -6014.484,E2 -6014.484} C_VEL
LIN {X 0,Y 495.561,Z 266.971,A -85,B 0,C 180,E1 -6017.451,E2 -6017.451} C_VEL
LIN {X 0,Y 497.322,Z 277.249,A -85,B 0,C 180,E1 -6017.647,E2 -6017.647} C_VEL
LIN {X 0,Y 496.943,Z 342.681,A -85,B 0,C 180,E1 -6018.606,E2 -6018.606} C_VEL
LIN {X 0,Y 496.845,Z 351.828,A -85,B 0,C 180,E1 -6018.836,E2 -6018.836} C_VEL
LIN {X 0,Y 496.708,Z 361.434,A -85,B 0,C 180,E1 -6019.194,E2 -6019.194} C_VEL
LIN {X 0,Y 496.555,Z 371.47,A -85,B 0,C 180,E1 -6019.706,E2 -6019.706} C_VEL
LIN {X 0,Y 496.35,Z 381.879,A -85,B 0,C 180,E1 -6020.423,E2 -6020.423} C_VEL
LIN {X 0,Y 496.045,Z 390.008,A -85,B 0,C 180,E1 -6021.136,E2 -6021.136} C_VEL
LIN {X 0,Y 495.852,Z 396.708,A -85,B 0,C 180,E1 -6021.851,E2 -6021.851} C_VEL
LIN {X 0,Y 495.662,Z 403.046,A -85,B 0,C 180,E1 -6022.668,E2 -6022.668} C_VEL
LIN {X 0,Y 495.521,Z 409.474,A -85,B 0,C 180,E1 -6023.689,E2 -6023.689} C_VEL
LIN {X 0,Y 495.298,Z 412.715,A -85,B 0,C 180,E1 -6024.299,E2 -6024.299} C_VEL
LIN {X 0,Y 495.363,Z 416.366,A -85,B 0,C 180,E1 -6025.116,E2 -6025.116} C_VEL
LIN {X 0,Y 495.213,Z 419.356,A -85,B 0,C 180,E1 -6025.931,E2 -6025.931} C_VEL
LIN {X 0,Y 495.233,Z 421.664,A -85,B 0,C 180,E1 -6026.745,E2 -6026.745} C_VEL
LIN {X 0,Y 495.074,Z 423.435,A -85,B 0,C 180,E1 -6027.559,E2 -6027.559} C_VEL
LIN {X 0,Y 494.97,Z 424.712,A -85,B 0,C 180,E1 -6028.372,E2 -6028.372} C_VEL
LIN {X 0,Y 494.931,Z 425.52,A -85,B 0,C 180,E1 -6029.186,E2 -6029.186} C_VEL
LIN {X 0,Y 494.927,Z 425.827,A -85,B 0,C 180,E1 -6030,E2 -6030} C_VEL
LIN {X 0,Y 494.932,Z 425.555,A -85,B 0,C 180,E1 -6030.813,E2 -6030.813} C_VEL
LIN {X 0,Y 494.971,Z 424.819,A -85,B 0,C 180,E1 -6031.627,E2 -6031.627} C_VEL
LIN {X 0,Y 495.074,Z 423.615,A -85,B 0,C 180,E1 -6032.44,E2 -6032.44} C_VEL
LIN {X 0,Y 495.231,Z 421.92,A -85,B 0,C 180,E1 -6033.254,E2 -6033.254} C_VEL
LIN {X 0,Y 495.27,Z 418.208,A -85,B 0,C 180,E1 -6034.476,E2 -6034.476} C_VEL
LIN {X 0,Y 495.295,Z 413.139,A -85,B 0,C 180,E1 -6035.7,E2 -6035.7} C_VEL
LIN {X 0,Y 495.583,Z 408.041,A -85,B 0,C 180,E1 -6036.653,E2 -6036.653} C_VEL
LIN {X 0,Y 495.736,Z 400.814,A -85,B 0,C 180,E1 -6037.74,E2 -6037.74} C_VEL
LIN {X 0,Y 495.982,Z 392.93,A -85,B 0,C 180,E1 -6038.659,E2 -6038.659} C_VEL
LIN {X 0,Y 496.229,Z 385.407,A -85,B 0,C 180,E1 -6039.373,E2 -6039.373} C_VEL
LIN {X 0,Y 496.362,Z 377.528,A -85,B 0,C 180,E1 -6039.988,E2 -6039.988} C_VEL
LIN {X 0,Y 496.582,Z 369.387,A -85,B 0,C 180,E1 -6040.498,E2 -6040.498} C_VEL
LIN {X 0,Y 496.762,Z 361.146,A -85,B 0,C 180,E1 -6040.907,E2 -6040.907} C_VEL
LIN {X 0,Y 496.833,Z 352.264,A -85,B 0,C 180,E1 -6041.241,E2 -6041.241} C_VEL
LIN {X 0,Y 497.007,Z 342.703,A -85,B 0,C 180,E1 -6041.482,E2 -6041.482} C_VEL
LIN {X 0,Y 497.133,Z 276.077,A -85,B 0,C 180,E1 -6042.465,E2 -6042.465} C_VEL
LIN {X 0,Y 495.558,Z 266.953,A -85,B 0,C 180,E1 -6042.645,E2 -6042.645} C_VEL
LIN {X 0,Y 495.563,Z 253.575,A -85,B 0,C 180,E1 -6045.631,E2 -6045.631} C_VEL
LIN {X 0,Y 495.772,Z 253.54,A -85,B 0,C 180,E1 -6048.234,E2 -6048.234} C_VEL
LIN {X 0,Y 495.772,Z 253.541,A -85,B 0,C 180,E1 -6050.756,E2 -6050.756} C_VEL
LIN {X 0,Y 495.732,Z 253.548,A -85,B 0,C 180,E1 -6053.387,E2 -6053.387} C_VEL
LIN {X 0,Y 495.715,Z 253.547,A -85,B 0,C 180,E1 -6056.072,E2 -6056.072} C_VEL
LIN {X 0,Y 495.716,Z 253.55,A -85,B 0,C 180,E1 -6058.818,E2 -6058.818} C_VEL
LIN {X 0,Y 495.735,Z 253.546,A -85,B 0,C 180,E1 -6061.721,E2 -6061.721} C_VEL
LIN {X 0,Y 495.754,Z 253.545,A -85,B 0,C 180,E1 -6064.691,E2 -6064.691} C_VEL
LIN {X 0,Y 495.716,Z 253.549,A -85,B 0,C 180,E1 -6067.562,E2 -6067.562} C_VEL
LIN {X 0,Y 495.739,Z 253.544,A -85,B 0,C 180,E1 -6070.044,E2 -6070.044} C_VEL
LIN {X 0,Y 495.691,Z 253.553,A -85,B 0,C 180,E1 -6072.886,E2 -6072.886} C_VEL
LIN {X 0,Y 495.718,Z 253.547,A -85,B 0,C 180,E1 -6075.997,E2 -6075.997} C_VEL
LIN {X 0,Y 495.721,Z 253.548,A -85,B 0,C 180,E1 -6079.295,E2 -6079.295} C_VEL
LIN {X 0,Y 495.722,Z 253.547,A -85,B 0,C 180,E1 -6081.406,E2 -6081.406} C_VEL
LIN {X 0,Y 495.734,Z 253.548,A -85,B 0,C 180,E1 -6084.461,E2 -6084.461} C_VEL
LIN {X 0,Y 495.745,Z 253.544,A -85,B 0,C 180,E1 -6087.404,E2 -6087.404} C_VEL
LIN {X 0,Y 495.735,Z 253.549,A -85,B 0,C 180,E1 -6090.251,E2 -6090.251} C_VEL
LIN {X 0,Y 495.733,Z 253.545,A -85,B 0,C 180,E1 -6093.27,E2 -6093.27} C_VEL
LIN {X 0,Y 495.704,Z 253.549,A -85,B 0,C 180,E1 -6095.722,E2 -6095.722} C_VEL
LIN {X 0,Y 495.727,Z 253.549,A -85,B 0,C 180,E1 -6098.37,E2 -6098.37} C_VEL
LIN {X 0,Y 495.758,Z 253.543,A -85,B 0,C 180,E1 -6100.97,E2 -6100.97} C_VEL
LIN {X 0,Y 495.797,Z 253.541,A -85,B 0,C 180,E1 -6104.558,E2 -6104.558} C_VEL
LIN {X 0,Y 495.816,Z 253.537,A -85,B 0,C 180,E1 -6107.969,E2 -6107.969} C_VEL
LIN {X 0,Y 495.788,Z 253.538,A -85,B 0,C 180,E1 -6111.029,E2 -6111.029} C_VEL
LIN {X 0,Y 495.816,Z 253.536,A -85,B 0,C 180,E1 -6113.489,E2 -6113.489} C_VEL
LIN {X 0,Y 495.698,Z 253.552,A -85,B 0,C 180,E1 -6115.935,E2 -6115.935} C_VEL
LIN {X 0,Y 495.969,Z 253.518,A -85,B 0,C 180,E1 -6117.563,E2 -6117.563} C_VEL
LIN {X 0,Y 495.966,Z 253.52,A -85,B 0,C 180,E1 -6120,E2 -6120} C_VEL
LIN {X 0,Y 495.969,Z 253.517,A -85,B 0,C 180,E1 -6122.436,E2 -6122.436} C_VEL
LIN {X 0,Y 495.844,Z 253.534,A -85,B 0,C 180,E1 -6125.694,E2 -6125.694} C_VEL
LIN {X 0,Y 495.804,Z 253.539,A -85,B 0,C 180,E1 -6128.149,E2 -6128.149} C_VEL
LIN {X 0,Y 495.815,Z 253.537,A -85,B 0,C 180,E1 -6131.446,E2 -6131.446} C_VEL
LIN {X 0,Y 495.768,Z 253.54,A -85,B 0,C 180,E1 -6134.783,E2 -6134.783} C_VEL
LIN {X 0,Y 495.741,Z 253.544,A -85,B 0,C 180,E1 -6138.226,E2 -6138.226} C_VEL
LIN {X 0,Y 495.74,Z 253.544,A -85,B 0,C 180,E1 -6140.758,E2 -6140.758} C_VEL
LIN {X 0,Y 495.724,Z 253.55,A -85,B 0,C 180,E1 -6143.388,E2 -6143.388} C_VEL
LIN {X 0,Y 495.732,Z 253.545,A -85,B 0,C 180,E1 -6146.729,E2 -6146.729} C_VEL
LIN {X 0,Y 495.689,Z 253.552,A -85,B 0,C 180,E1 -6149.751,E2 -6149.751} C_VEL
LIN {X 0,Y 495.742,Z 253.544,A -85,B 0,C 180,E1 -6152.596,E2 -6152.596} C_VEL
LIN {X 0,Y 495.723,Z 253.548,A -85,B 0,C 180,E1 -6155.54,E2 -6155.54} C_VEL
LIN {X 0,Y 495.732,Z 253.546,A -85,B 0,C 180,E1 -6158.765,E2 -6158.765} C_VEL
LIN {X 0,Y 495.717,Z 253.546,A -85,B 0,C 180,E1 -6161.785,E2 -6161.785} C_VEL
LIN {X 0,Y 495.728,Z 253.55,A -85,B 0,C 180,E1 -6165.142,E2 -6165.142} C_VEL
LIN {X 0,Y 495.718,Z 253.546,A -85,B 0,C 180,E1 -6168.216,E2 -6168.216} C_VEL
LIN {X 0,Y 495.733,Z 253.546,A -85,B 0,C 180,E1 -6171.236,E2 -6171.236} C_VEL
LIN {X 0,Y 495.722,Z 253.548,A -85,B 0,C 180,E1 -6174.461,E2 -6174.461} C_VEL
LIN {X 0,Y 495.72,Z 253.545,A -85,B 0,C 180,E1 -6177.403,E2 -6177.403} C_VEL
LIN {X 0,Y 495.691,Z 253.551,A -85,B 0,C 180,E1 -6180.249,E2 -6180.249} C_VEL
LIN {X 0,Y 495.717,Z 253.548,A -85,B 0,C 180,E1 -6183.275,E2 -6183.275} C_VEL
LIN {X 0,Y 495.759,Z 253.563,A -85,B 0,C 180,E1 -6185.782,E2 -6185.782} C_VEL
LIN {X 0,Y 496.935,Z 261.213,A -85,B 0,C 180,E1 -6187.214,E2 -6187.214} C_VEL
LIN {X 0,Y 496.537,Z 276.46,A -85,B 0,C 180,E1 -6189.926,E2 -6189.926} C_VEL
LIN {X 0,Y 496.211,Z 290.999,A -85,B 0,C 180,E1 -6192.485,E2 -6192.485} C_VEL
LIN {X 0,Y 495.835,Z 309.103,A -85,B 0,C 180,E1 -6195.639,E2 -6195.639} C_VEL
LIN {X 0,Y 495.582,Z 319.153,A -85,B 0,C 180,E1 -6197.377,E2 -6197.377} C_VEL
LIN {X 0,Y 497.126,Z 334.06,A -85,B 0,C 180,E1 -6197.643,E2 -6197.643} C_VEL
LIN {X 0,Y 496.824,Z 397.473,A -85,B 0,C 180,E1 -6198.578,E2 -6198.578} C_VEL
LIN {X 0,Y 496.593,Z 407.947,A -85,B 0,C 180,E1 -6198.857,E2 -6198.857} C_VEL
LIN {X 0,Y 496.419,Z 418.679,A -85,B 0,C 180,E1 -6199.292,E2 -6199.292} C_VEL
LIN {X 0,Y 496.094,Z 429.33,A -85,B 0,C 180,E1 -6199.904,E2 -6199.904} C_VEL
LIN {X 0,Y 495.944,Z 437.682,A -85,B 0,C 180,E1 -6200.518,E2 -6200.518} C_VEL
LIN {X 0,Y 495.675,Z 445.584,A -85,B 0,C 180,E1 -6201.233,E2 -6201.233} C_VEL
LIN {X 0,Y 495.445,Z 452.977,A -85,B 0,C 180,E1 -6202.051,E2 -6202.051} C_VEL
LIN {X 0,Y 495.324,Z 460.489,A -85,B 0,C 180,E1 -6203.074,E2 -6203.074} C_VEL
LIN {X 0,Y 495.186,Z 467.347,A -85,B 0,C 180,E1 -6204.299,E2 -6204.299} C_VEL
LIN {X 0,Y 495.048,Z 472.553,A -85,B 0,C 180,E1 -6205.522,E2 -6205.522} C_VEL
LIN {X 0,Y 495.094,Z 475.221,A -85,B 0,C 180,E1 -6206.338,E2 -6206.338} C_VEL
LIN {X 0,Y 495.056,Z 478.144,A -85,B 0,C 180,E1 -6207.56,E2 -6207.56} C_VEL
LIN {X 0,Y 494.962,Z 479.401,A -85,B 0,C 180,E1 -6208.373,E2 -6208.373} C_VEL
LIN {X 0,Y 494.919,Z 480.184,A -85,B 0,C 180,E1 -6209.187,E2 -6209.187} C_VEL
LIN {X 0,Y 494.916,Z 480.481,A -85,B 0,C 180,E1 -6210,E2 -6210} C_VEL
LIN {X 0,Y 494.919,Z 480.183,A -85,B 0,C 180,E1 -6210.814,E2 -6210.814} C_VEL
LIN {X 0,Y 494.962,Z 479.399,A -85,B 0,C 180,E1 -6211.628,E2 -6211.628} C_VEL
LIN {X 0,Y 495.056,Z 478.141,A -85,B 0,C 180,E1 -6212.441,E2 -6212.441} C_VEL
LIN {X 0,Y 495.094,Z 475.218,A -85,B 0,C 180,E1 -6213.663,E2 -6213.663} C_VEL
LIN {X 0,Y 495.048,Z 472.549,A -85,B 0,C 180,E1 -6214.479,E2 -6214.479} C_VEL
LIN {X 0,Y 495.187,Z 467.34,A -85,B 0,C 180,E1 -6215.702,E2 -6215.702} C_VEL
LIN {X 0,Y 495.29,Z 460.744,A -85,B 0,C 180,E1 -6216.887,E2 -6216.887} C_VEL
LIN {X 0,Y 495.446,Z 452.972,A -85,B 0,C 180,E1 -6217.95,E2 -6217.95} C_VEL
LIN {X 0,Y 495.676,Z 445.583,A -85,B 0,C 180,E1 -6218.768,E2 -6218.768} C_VEL
LIN {X 0,Y 495.945,Z 437.675,A -85,B 0,C 180,E1 -6219.482,E2 -6219.482} C_VEL
LIN {X 0,Y 496.095,Z 429.318,A -85,B 0,C 180,E1 -6220.097,E2 -6220.097} C_VEL
LIN {X 0,Y 496.409,Z 418.664,A -85,B 0,C 180,E1 -6220.709,E2 -6220.709} C_VEL
LIN {X 0,Y 496.603,Z 407.089,A -85,B 0,C 180,E1 -6221.17,E2 -6221.17} C_VEL
LIN {X 0,Y 496.82,Z 397.428,A -85,B 0,C 180,E1 -6221.423,E2 -6221.423} C_VEL
LIN {X 0,Y 497.129,Z 334.987,A -85,B 0,C 180,E1 -6222.343,E2 -6222.343} C_VEL
LIN {X 0,Y 495.581,Z 319.124,A -85,B 0,C 180,E1 -6222.628,E2 -6222.628} C_VEL
LIN {X 0,Y 495.844,Z 304.687,A -85,B 0,C 180,E1 -6225.13,E2 -6225.13} C_VEL
LIN {X 0,Y 496.292,Z 287.361,A -85,B 0,C 180,E1 -6228.153,E2 -6228.153} C_VEL
LIN {X 0,Y 496.72,Z 270.014,A -85,B 0,C 180,E1 -6231.214,E2 -6231.214} C_VEL
LIN {X 0,Y 496.94,Z 261.2,A -85,B 0,C 180,E1 -6232.787,E2 -6232.787} C_VEL
LIN {X 0,Y 495.783,Z 253.54,A -85,B 0,C 180,E1 -6234.246,E2 -6234.246} C_VEL
LIN {X 0,Y 495.717,Z 253.55,A -85,B 0,C 180,E1 -6236.98,E2 -6236.98} C_VEL
LIN {X 0,Y 495.695,Z 253.55,A -85,B 0,C 180,E1 -6239.751,E2 -6239.751} C_VEL
LIN {X 0,Y 495.724,Z 253.545,A -85,B 0,C 180,E1 -6242.598,E2 -6242.598} C_VEL
LIN {X 0,Y 495.718,Z 253.548,A -85,B 0,C 180,E1 -6245.541,E2 -6245.541} C_VEL
LIN {X 0,Y 495.725,Z 253.547,A -85,B 0,C 180,E1 -6248.763,E2 -6248.763} C_VEL
LIN {X 0,Y 495.7,Z 253.548,A -85,B 0,C 180,E1 -6251.787,E2 -6251.787} C_VEL
LIN {X 0,Y 495.731,Z 253.549,A -85,B 0,C 180,E1 -6255.142,E2 -6255.142} C_VEL
LIN {X 0,Y 495.722,Z 253.545,A -85,B 0,C 180,E1 -6258.215,E2 -6258.215} C_VEL
LIN {X 0,Y 495.716,Z 253.548,A -85,B 0,C 180,E1 -6261.405,E2 -6261.405} C_VEL
LIN {X 0,Y 495.725,Z 253.548,A -85,B 0,C 180,E1 -6264.461,E2 -6264.461} C_VEL
LIN {X 0,Y 495.724,Z 253.546,A -85,B 0,C 180,E1 -6267.403,E2 -6267.403} C_VEL
LIN {X 0,Y 495.695,Z 253.551,A -85,B 0,C 180,E1 -6270.249,E2 -6270.249} C_VEL
LIN {X 0,Y 495.721,Z 253.547,A -85,B 0,C 180,E1 -6273.275,E2 -6273.275} C_VEL
LIN {X 0,Y 495.696,Z 253.549,A -85,B 0,C 180,E1 -6275.722,E2 -6275.722} C_VEL
LIN {X 0,Y 495.723,Z 253.551,A -85,B 0,C 180,E1 -6278.37,E2 -6278.37} C_VEL
LIN {X 0,Y 495.748,Z 253.543,A -85,B 0,C 180,E1 -6281.774,E2 -6281.774} C_VEL
LIN {X 0,Y 495.744,Z 253.543,A -85,B 0,C 180,E1 -6285.216,E2 -6285.216} C_VEL
LIN {X 0,Y 495.814,Z 253.537,A -85,B 0,C 180,E1 -6288.554,E2 -6288.554} C_VEL
LIN {X 0,Y 495.811,Z 253.538,A -85,B 0,C 180,E1 -6291.851,E2 -6291.851} C_VEL
LIN {X 0,Y 495.85,Z 253.534,A -85,B 0,C 180,E1 -6294.306,E2 -6294.306} C_VEL
LIN {X 0,Y 495.975,Z 253.516,A -85,B 0,C 180,E1 -6297.564,E2 -6297.564} C_VEL
LIN {X 0,Y 495.972,Z 253.519,A -85,B 0,C 180,E1 -6300,E2 -6300} C_VEL
LIN {X 0,Y 495.975,Z 253.517,A -85,B 0,C 180,E1 -6302.436,E2 -6302.436} C_VEL
LIN {X 0,Y 495.85,Z 253.534,A -85,B 0,C 180,E1 -6305.694,E2 -6305.694} C_VEL
LIN {X 0,Y 495.811,Z 253.538,A -85,B 0,C 180,E1 -6308.149,E2 -6308.149} C_VEL
LIN {X 0,Y 495.822,Z 253.536,A -85,B 0,C 180,E1 -6311.446,E2 -6311.446} C_VEL
LIN {X 0,Y 495.776,Z 253.539,A -85,B 0,C 180,E1 -6314.783,E2 -6314.783} C_VEL
LIN {X 0,Y 495.748,Z 253.545,A -85,B 0,C 180,E1 -6318.226,E2 -6318.226} C_VEL
LIN {X 0,Y 495.747,Z 253.543,A -85,B 0,C 180,E1 -6320.758,E2 -6320.758} C_VEL
LIN {X 0,Y 495.735,Z 253.549,A -85,B 0,C 180,E1 -6323.388,E2 -6323.388} C_VEL
LIN {X 0,Y 495.718,Z 253.549,A -85,B 0,C 180,E1 -6326.072,E2 -6326.072} C_VEL
LIN {X 0,Y 495.716,Z 253.548,A -85,B 0,C 180,E1 -6328.818,E2 -6328.818} C_VEL
LIN {X 0,Y 495.75,Z 253.546,A -85,B 0,C 180,E1 -6331.724,E2 -6331.724} C_VEL
LIN {X 0,Y 495.758,Z 253.542,A -85,B 0,C 180,E1 -6334.692,E2 -6334.692} C_VEL
LIN {X 0,Y 495.713,Z 253.551,A -85,B 0,C 180,E1 -6337.563,E2 -6337.563} C_VEL
LIN {X 0,Y 495.743,Z 253.544,A -85,B 0,C 180,E1 -6340.045,E2 -6340.045} C_VEL
LIN {X 0,Y 495.696,Z 253.553,A -85,B 0,C 180,E1 -6342.886,E2 -6342.886} C_VEL
LIN {X 0,Y 495.723,Z 253.546,A -85,B 0,C 180,E1 -6345.998,E2 -6345.998} C_VEL
LIN {X 0,Y 495.728,Z 253.55,A -85,B 0,C 180,E1 -6349.296,E2 -6349.296} C_VEL
LIN {X 0,Y 495.746,Z 253.547,A -85,B 0,C 180,E1 -6351.408,E2 -6351.408} C_VEL
LIN {X 0,Y 495.744,Z 253.545,A -85,B 0,C 180,E1 -6354.462,E2 -6354.462} C_VEL
LIN {X 0,Y 495.749,Z 253.545,A -85,B 0,C 180,E1 -6357.404,E2 -6357.404} C_VEL
LIN {X 0,Y 495.715,Z 253.547,A -85,B 0,C 180,E1 -6360.713,E2 -6360.713} C_VEL
LIN {X 0,Y 495.04,Z 253.635,A -85,B 0,C 180,E1 -6361.392,E2 -6361.392} C_VEL
LIN {X 0,Y 492.17,Z 253.991,A -85,B 0,C 180,E1 -6362.494,E2 -6362.494} C_VEL
LIN {X 0,Y 489.762,Z 254.29,A -85,B 0,C 180,E1 -6363.382,E2 -6363.382} C_VEL
LIN {X 0,Y 488.752,Z 254.415,A -85,B 0,C 180,E1 -6364.068,E2 -6364.068} C_VEL
LIN {X 0,Y 488.682,Z 254.424,A -85,B 0,C 180,E1 -6364.3,E2 -6364.3} C_VEL
LIN {X 0,Y 488.71,Z 254.423,A -85,B 0,C 180,E1 -6367.152,E2 -6367.152} C_VEL
LIN {X 0,Y 488.72,Z 254.418,A -85,B 0,C 180,E1 -6369.81,E2 -6369.81} C_VEL
LIN {X 0,Y 488.681,Z 254.428,A -85,B 0,C 180,E1 -6372.421,E2 -6372.421} C_VEL
LIN {X 0,Y 488.559,Z 254.575,A -85,B 0,C 180,E1 -6374.435,E2 -6374.435} C_VEL
LIN {X 0,Y 488.529,Z 267.283,A -85,B 0,C 180,E1 -6377.263,E2 -6377.263} C_VEL
LIN {X 0,Y 490.409,Z 278.657,A -85,B 0,C 180,E1 -6377.485,E2 -6377.485} C_VEL
LIN {X 0,Y 490,Z 343.097,A -85,B 0,C 180,E1 -6378.442,E2 -6378.442} C_VEL
LIN {X 0,Y 489.896,Z 352.235,A -85,B 0,C 180,E1 -6378.675,E2 -6378.675} C_VEL
LIN {X 0,Y 489.753,Z 361.837,A -85,B 0,C 180,E1 -6379.039,E2 -6379.039} C_VEL
LIN {X 0,Y 489.582,Z 371.87,A -85,B 0,C 180,E1 -6379.558,E2 -6379.558} C_VEL
LIN {X 0,Y 489.375,Z 382.275,A -85,B 0,C 180,E1 -6380.285,E2 -6380.285} C_VEL
LIN {X 0,Y 489.058,Z 390.404,A -85,B 0,C 180,E1 -6381.009,E2 -6381.009} C_VEL
LIN {X 0,Y 488.832,Z 397.103,A -85,B 0,C 180,E1 -6381.733,E2 -6381.733} C_VEL
LIN {X 0,Y 488.652,Z 403.44,A -85,B 0,C 180,E1 -6382.562,E2 -6382.562} C_VEL
LIN {X 0,Y 488.54,Z 408.703,A -85,B 0,C 180,E1 -6383.391,E2 -6383.391} C_VEL
LIN {X 0,Y 488.259,Z 413.108,A -85,B 0,C 180,E1 -6384.217,E2 -6384.217} C_VEL
LIN {X 0,Y 488.314,Z 416.759,A -85,B 0,C 180,E1 -6385.046,E2 -6385.046} C_VEL
LIN {X 0,Y 488.16,Z 419.748,A -85,B 0,C 180,E1 -6385.872,E2 -6385.872} C_VEL
LIN {X 0,Y 488.163,Z 422.057,A -85,B 0,C 180,E1 -6386.698,E2 -6386.698} C_VEL
LIN {X 0,Y 488.014,Z 423.826,A -85,B 0,C 180,E1 -6387.523,E2 -6387.523} C_VEL
LIN {X 0,Y 487.9,Z 425.103,A -85,B 0,C 180,E1 -6388.349,E2 -6388.349} C_VEL
LIN {X 0,Y 487.853,Z 425.911,A -85,B 0,C 180,E1 -6389.174,E2 -6389.174} C_VEL
LIN {X 0,Y 487.846,Z 426.218,A -85,B 0,C 180,E1 -6390,E2 -6390} C_VEL
LIN {X 0,Y 487.854,Z 425.946,A -85,B 0,C 180,E1 -6390.825,E2 -6390.825} C_VEL
LIN {X 0,Y 487.9,Z 425.209,A -85,B 0,C 180,E1 -6391.65,E2 -6391.65} C_VEL
LIN {X 0,Y 488.014,Z 424.004,A -85,B 0,C 180,E1 -6392.476,E2 -6392.476} C_VEL
LIN {X 0,Y 488.169,Z 421.17,A -85,B 0,C 180,E1 -6393.714,E2 -6393.714} C_VEL
LIN {X 0,Y 488.219,Z 418.597,A -85,B 0,C 180,E1 -6394.541,E2 -6394.541} C_VEL
LIN {X 0,Y 488.255,Z 413.528,A -85,B 0,C 180,E1 -6395.782,E2 -6395.782} C_VEL
LIN {X 0,Y 488.571,Z 407.821,A -85,B 0,C 180,E1 -6396.857,E2 -6396.857} C_VEL
LIN {X 0,Y 488.71,Z 401.201,A -85,B 0,C 180,E1 -6397.852,E2 -6397.852} C_VEL
LIN {X 0,Y 488.972,Z 393.317,A -85,B 0,C 180,E1 -6398.784,E2 -6398.784} C_VEL
LIN {X 0,Y 489.245,Z 385.792,A -85,B 0,C 180,E1 -6399.508,E2 -6399.508} C_VEL
LIN {X 0,Y 489.378,Z 377.912,A -85,B 0,C 180,E1 -6400.132,E2 -6400.132} C_VEL
LIN {X 0,Y 489.626,Z 369.768,A -85,B 0,C 180,E1 -6400.649,E2 -6400.649} C_VEL
LIN {X 0,Y 489.824,Z 361.525,A -85,B 0,C 180,E1 -6401.063,E2 -6401.063} C_VEL
LIN {X 0,Y 489.89,Z 352.64,A -85,B 0,C 180,E1 -6401.402,E2 -6401.402} C_VEL
LIN {X 0,Y 490.082,Z 343.214,A -85,B 0,C 180,E1 -6401.644,E2 -6401.644} C_VEL
LIN {X 0,Y 490.273,Z 277.163,A -85,B 0,C 180,E1 -6402.631,E2 -6402.631} C_VEL
LIN {X 0,Y 488.535,Z 267.309,A -85,B 0,C 180,E1 -6402.824,E2 -6402.824} C_VEL
LIN {X 0,Y 488.531,Z 254.451,A -85,B 0,C 180,E1 -6405.695,E2 -6405.695} C_VEL
LIN {X 0,Y 488.743,Z 254.415,A -85,B 0,C 180,E1 -6408.442,E2 -6408.442} C_VEL
LIN {X 0,Y 488.703,Z 254.425,A -85,B 0,C 180,E1 -6411.07,E2 -6411.07} C_VEL
LIN {X 0,Y 488.663,Z 254.428,A -85,B 0,C 180,E1 -6413.746,E2 -6413.746} C_VEL
LIN {X 0,Y 488.68,Z 254.424,A -85,B 0,C 180,E1 -6416.476,E2 -6416.476} C_VEL
LIN {X 0,Y 488.686,Z 254.426,A -85,B 0,C 180,E1 -6419.272,E2 -6419.272} C_VEL
LIN {X 0,Y 488.687,Z 254.422,A -85,B 0,C 180,E1 -6422.148,E2 -6422.148} C_VEL
LIN {X 0,Y 488.707,Z 254.423,A -85,B 0,C 180,E1 -6425.115,E2 -6425.115} C_VEL
LIN {X 0,Y 488.671,Z 254.425,A -85,B 0,C 180,E1 -6428.2,E2 -6428.2} C_VEL
LIN {X 0,Y 488.69,Z 254.423,A -85,B 0,C 180,E1 -6430.341,E2 -6430.341} C_VEL
LIN {X 0,Y 488.669,Z 254.425,A -85,B 0,C 180,E1 -6433.656,E2 -6433.656} C_VEL
LIN {X 0,Y 488.669,Z 254.427,A -85,B 0,C 180,E1 -6436.343,E2 -6436.343} C_VEL
LIN {X 0,Y 488.699,Z 254.421,A -85,B 0,C 180,E1 -6439.673,E2 -6439.673} C_VEL
LIN {X 0,Y 488.66,Z 254.429,A -85,B 0,C 180,E1 -6442.839,E2 -6442.839} C_VEL
LIN {X 0,Y 488.712,Z 254.42,A -85,B 0,C 180,E1 -6445.886,E2 -6445.886} C_VEL
LIN {X 0,Y 488.677,Z 254.427,A -85,B 0,C 180,E1 -6448.819,E2 -6448.819} C_VEL
LIN {X 0,Y 488.686,Z 254.423,A -85,B 0,C 180,E1 -6451.667,E2 -6451.667} C_VEL
LIN {X 0,Y 488.684,Z 254.426,A -85,B 0,C 180,E1 -6454.441,E2 -6454.441} C_VEL
LIN {X 0,Y 488.701,Z 254.421,A -85,B 0,C 180,E1 -6457.152,E2 -6457.152} C_VEL
LIN {X 0,Y 488.71,Z 254.422,A -85,B 0,C 180,E1 -6459.81,E2 -6459.81} C_VEL
LIN {X 0,Y 488.676,Z 254.428,A -85,B 0,C 180,E1 -6462.421,E2 -6462.421} C_VEL
LIN {X 0,Y 488.74,Z 254.416,A -85,B 0,C 180,E1 -6464.999,E2 -6464.999} C_VEL
LIN {X 0,Y 488.778,Z 254.416,A -85,B 0,C 180,E1 -6468.387,E2 -6468.387} C_VEL
LIN {X 0,Y 488.751,Z 254.417,A -85,B 0,C 180,E1 -6471.732,E2 -6471.732} C_VEL
LIN {X 0,Y 488.808,Z 254.412,A -85,B 0,C 180,E1 -6474.224,E2 -6474.224} C_VEL
LIN {X 0,Y 488.935,Z 254.394,A -85,B 0,C 180,E1 -6477.528,E2 -6477.528} C_VEL
LIN {X 0,Y 488.935,Z 254.396,A -85,B 0,C 180,E1 -6480,E2 -6480} C_VEL
LIN {X 0,Y 488.935,Z 254.393,A -85,B 0,C 180,E1 -6482.471,E2 -6482.471} C_VEL
LIN {X 0,Y 488.804,Z 254.411,A -85,B 0,C 180,E1 -6485.776,E2 -6485.776} C_VEL
LIN {X 0,Y 488.75,Z 254.416,A -85,B 0,C 180,E1 -6488.267,E2 -6488.267} C_VEL
LIN {X 0,Y 488.778,Z 254.414,A -85,B 0,C 180,E1 -6491.613,E2 -6491.613} C_VEL
LIN {X 0,Y 488.74,Z 254.417,A -85,B 0,C 180,E1 -6495.001,E2 -6495.001} C_VEL
LIN {X 0,Y 488.699,Z 254.42,A -85,B 0,C 180,E1 -6498.444,E2 -6498.444} C_VEL
LIN {X 0,Y 488.683,Z 254.424,A -85,B 0,C 180,E1 -6501.072,E2 -6501.072} C_VEL
LIN {X 0,Y 488.654,Z 254.43,A -85,B 0,C 180,E1 -6503.747,E2 -6503.747} C_VEL
LIN {X 0,Y 488.675,Z 254.423,A -85,B 0,C 180,E1 -6506.477,E2 -6506.477} C_VEL
LIN {X 0,Y 488.653,Z 254.431,A -85,B 0,C 180,E1 -6509.275,E2 -6509.275} C_VEL
LIN {X 0,Y 488.684,Z 254.422,A -85,B 0,C 180,E1 -6512.148,E2 -6512.148} C_VEL
LIN {X 0,Y 488.7,Z 254.425,A -85,B 0,C 180,E1 -6515.116,E2 -6515.116} C_VEL
LIN {X 0,Y 488.649,Z 254.426,A -85,B 0,C 180,E1 -6518.203,E2 -6518.203} C_VEL
LIN {X 0,Y 488.688,Z 254.422,A -85,B 0,C 180,E1 -6520.341,E2 -6520.341} C_VEL
LIN {X 0,Y 488.668,Z 254.424,A -85,B 0,C 180,E1 -6523.656,E2 -6523.656} C_VEL
LIN {X 0,Y 488.66,Z 254.426,A -85,B 0,C 180,E1 -6526.343,E2 -6526.343} C_VEL
LIN {X 0,Y 488.699,Z 254.42,A -85,B 0,C 180,E1 -6529.674,E2 -6529.674} C_VEL
LIN {X 0,Y 488.644,Z 254.434,A -85,B 0,C 180,E1 -6532.839,E2 -6532.839} C_VEL
LIN {X 0,Y 488.703,Z 254.419,A -85,B 0,C 180,E1 -6535.886,E2 -6535.886} C_VEL
LIN {X 0,Y 488.654,Z 254.431,A -85,B 0,C 180,E1 -6538.818,E2 -6538.818} C_VEL
LIN {X 0,Y 488.68,Z 254.423,A -85,B 0,C 180,E1 -6541.668,E2 -6541.668} C_VEL
LIN {X 0,Y 488.687,Z 254.427,A -85,B 0,C 180,E1 -6544.962,E2 -6544.962} C_VEL
LIN {X 0,Y 488.744,Z 254.541,A -85,B 0,C 180,E1 -6545.666,E2 -6545.666} C_VEL
LIN {X 0,Y 489.967,Z 262.7,A -85,B 0,C 180,E1 -6547.215,E2 -6547.215} C_VEL
LIN {X 0,Y 489.519,Z 278.499,A -85,B 0,C 180,E1 -6550.064,E2 -6550.064} C_VEL
LIN {X 0,Y 489.122,Z 293.027,A -85,B 0,C 180,E1 -6552.654,E2 -6552.654} C_VEL
LIN {X 0,Y 488.709,Z 311.117,A -85,B 0,C 180,E1 -6555.85,E2 -6555.85} C_VEL
LIN {X 0,Y 488.553,Z 318.834,A -85,B 0,C 180,E1 -6557.205,E2 -6557.205} C_VEL
LIN {X 0,Y 490.184,Z 333.678,A -85,B 0,C 180,E1 -6557.465,E2 -6557.465} C_VEL
LIN {X 0,Y 489.878,Z 396.071,A -85,B 0,C 180,E1 -6558.393,E2 -6558.393} C_VEL
LIN {X 0,Y 489.738,Z 405.065,A -85,B 0,C 180,E1 -6558.62,E2 -6558.62} C_VEL
LIN {X 0,Y 489.49,Z 413.55,A -85,B 0,C 180,E1 -6558.929,E2 -6558.929} C_VEL
LIN {X 0,Y 489.288,Z 422.08,A -85,B 0,C 180,E1 -6559.343,E2 -6559.343} C_VEL
LIN {X 0,Y 489.036,Z 430.445,A -85,B 0,C 180,E1 -6559.861,E2 -6559.861} C_VEL
LIN {X 0,Y 488.865,Z 438.524,A -85,B 0,C 180,E1 -6560.484,E2 -6560.484} C_VEL
LIN {X 0,Y 488.604,Z 446.218,A -85,B 0,C 180,E1 -6561.21,E2 -6561.21} C_VEL
LIN {X 0,Y 488.349,Z 454.294,A -85,B 0,C 180,E1 -6562.143,E2 -6562.143} C_VEL
LIN {X 0,Y 488.204,Z 461.353,A -85,B 0,C 180,E1 -6563.18,E2 -6563.18} C_VEL
LIN {X 0,Y 488.088,Z 466.953,A -85,B 0,C 180,E1 -6564.216,E2 -6564.216} C_VEL
LIN {X 0,Y 487.957,Z 472.16,A -85,B 0,C 180,E1 -6565.457,E2 -6565.457} C_VEL
LIN {X 0,Y 488.016,Z 474.829,A -85,B 0,C 180,E1 -6566.285,E2 -6566.285} C_VEL
LIN {X 0,Y 487.961,Z 477.751,A -85,B 0,C 180,E1 -6567.524,E2 -6567.524} C_VEL
LIN {X 0,Y 487.891,Z 479.01,A -85,B 0,C 180,E1 -6568.35,E2 -6568.35} C_VEL
LIN {X 0,Y 487.841,Z 479.793,A -85,B 0,C 180,E1 -6569.175,E2 -6569.175} C_VEL
LIN {X 0,Y 487.836,Z 480.09,A -85,B 0,C 180,E1 -6570,E2 -6570} C_VEL
LIN {X 0,Y 487.841,Z 479.793,A -85,B 0,C 180,E1 -6570.826,E2 -6570.826} C_VEL
LIN {X 0,Y 487.892,Z 479.008,A -85,B 0,C 180,E1 -6571.651,E2 -6571.651} C_VEL
LIN {X 0,Y 487.962,Z 477.749,A -85,B 0,C 180,E1 -6572.477,E2 -6572.477} C_VEL
LIN {X 0,Y 488.017,Z 474.826,A -85,B 0,C 180,E1 -6573.716,E2 -6573.716} C_VEL
LIN {X 0,Y 487.958,Z 472.156,A -85,B 0,C 180,E1 -6574.544,E2 -6574.544} C_VEL
LIN {X 0,Y 488.088,Z 466.946,A -85,B 0,C 180,E1 -6575.785,E2 -6575.785} C_VEL
LIN {X 0,Y 488.241,Z 460.081,A -85,B 0,C 180,E1 -6577.028,E2 -6577.028} C_VEL
LIN {X 0,Y 488.401,Z 452.579,A -85,B 0,C 180,E1 -6578.066,E2 -6578.066} C_VEL
LIN {X 0,Y 488.644,Z 445.189,A -85,B 0,C 180,E1 -6578.895,E2 -6578.895} C_VEL
LIN {X 0,Y 488.908,Z 437.28,A -85,B 0,C 180,E1 -6579.62,E2 -6579.62} C_VEL
LIN {X 0,Y 489.084,Z 428.923,A -85,B 0,C 180,E1 -6580.243,E2 -6580.243} C_VEL
LIN {X 0,Y 489.448,Z 418.271,A -85,B 0,C 180,E1 -6580.863,E2 -6580.863} C_VEL
LIN {X 0,Y 489.645,Z 406.693,A -85,B 0,C 180,E1 -6581.33,E2 -6581.33} C_VEL
LIN {X 0,Y 489.875,Z 397.029,A -85,B 0,C 180,E1 -6581.587,E2 -6581.587} C_VEL
LIN {X 0,Y 490.196,Z 337.833,A -85,B 0,C 180,E1 -6582.473,E2 -6582.473} C_VEL
LIN {X 0,Y 489.879,Z 331.221,A -85,B 0,C 180,E1 -6582.578,E2 -6582.578} C_VEL
LIN {X 0,Y 488.56,Z 318.765,A -85,B 0,C 180,E1 -6582.806,E2 -6582.806} C_VEL
LIN {X 0,Y 488.797,Z 304.639,A -85,B 0,C 180,E1 -6585.292,E2 -6585.292} C_VEL
LIN {X 0,Y 489.355,Z 286.069,A -85,B 0,C 180,E1 -6588.581,E2 -6588.581} C_VEL
LIN {X 0,Y 489.843,Z 267.555,A -85,B 0,C 180,E1 -6591.903,E2 -6591.903} C_VEL
LIN {X 0,Y 489.874,Z 261.341,A -85,B 0,C 180,E1 -6593.035,E2 -6593.035} C_VEL
LIN {X 0,Y 488.728,Z 254.418,A -85,B 0,C 180,E1 -6594.364,E2 -6594.364} C_VEL
LIN {X 0,Y 488.674,Z 254.43,A -85,B 0,C 180,E1 -6597.401,E2 -6597.401} C_VEL
LIN {X 0,Y 488.651,Z 254.425,A -85,B 0,C 180,E1 -6600.351,E2 -6600.351} C_VEL
LIN {X 0,Y 488.692,Z 254.425,A -85,B 0,C 180,E1 -6603.477,E2 -6603.477} C_VEL
LIN {X 0,Y 488.64,Z 254.426,A -85,B 0,C 180,E1 -6606.348,E2 -6606.348} C_VEL
LIN {X 0,Y 488.668,Z 254.429,A -85,B 0,C 180,E1 -6609.258,E2 -6609.258} C_VEL
LIN {X 0,Y 488.647,Z 254.427,A -85,B 0,C 180,E1 -6612.531,E2 -6612.531} C_VEL
LIN {X 0,Y 488.695,Z 254.424,A -85,B 0,C 180,E1 -6615.197,E2 -6615.197} C_VEL
LIN {X 0,Y 488.658,Z 254.428,A -85,B 0,C 180,E1 -6618.579,E2 -6618.579} C_VEL
LIN {X 0,Y 488.65,Z 254.426,A -85,B 0,C 180,E1 -6621.797,E2 -6621.797} C_VEL
LIN {X 0,Y 488.708,Z 254.422,A -85,B 0,C 180,E1 -6625.056,E2 -6625.056} C_VEL
LIN {X 0,Y 488.682,Z 254.423,A -85,B 0,C 180,E1 -6628.05,E2 -6628.05} C_VEL
LIN {X 0,Y 488.66,Z 254.426,A -85,B 0,C 180,E1 -6631.32,E2 -6631.32} C_VEL
LIN {X 0,Y 488.667,Z 254.424,A -85,B 0,C 180,E1 -6633.523,E2 -6633.523} C_VEL
LIN {X 0,Y 488.656,Z 254.429,A -85,B 0,C 180,E1 -6636.253,E2 -6636.253} C_VEL
LIN {X 0,Y 488.672,Z 254.425,A -85,B 0,C 180,E1 -6639.199,E2 -6639.199} C_VEL
LIN {X 0,Y 488.706,Z 254.42,A -85,B 0,C 180,E1 -6641.648,E2 -6641.648} C_VEL
LIN {X 0,Y 488.714,Z 254.42,A -85,B 0,C 180,E1 -6644.998,E2 -6644.998} C_VEL
LIN {X 0,Y 488.775,Z 254.415,A -85,B 0,C 180,E1 -6648.387,E2 -6648.387} C_VEL
LIN {X 0,Y 488.754,Z 254.416,A -85,B 0,C 180,E1 -6651.733,E2 -6651.733} C_VEL
LIN {X 0,Y 488.81,Z 254.411,A -85,B 0,C 180,E1 -6654.224,E2 -6654.224} C_VEL
LIN {X 0,Y 488.941,Z 254.392,A -85,B 0,C 180,E1 -6657.529,E2 -6657.529} C_VEL
LIN {X 0,Y 488.941,Z 254.395,A -85,B 0,C 180,E1 -6660,E2 -6660} C_VEL
LIN {X 0,Y 488.941,Z 254.393,A -85,B 0,C 180,E1 -6662.472,E2 -6662.472} C_VEL
LIN {X 0,Y 488.81,Z 254.412,A -85,B 0,C 180,E1 -6665.776,E2 -6665.776} C_VEL
LIN {X 0,Y 488.755,Z 254.417,A -85,B 0,C 180,E1 -6668.268,E2 -6668.268} C_VEL
LIN {X 0,Y 488.785,Z 254.415,A -85,B 0,C 180,E1 -6671.613,E2 -6671.613} C_VEL
LIN {X 0,Y 488.747,Z 254.415,A -85,B 0,C 180,E1 -6675.001,E2 -6675.001} C_VEL
LIN {X 0,Y 488.707,Z 254.421,A -85,B 0,C 180,E1 -6678.444,E2 -6678.444} C_VEL
LIN {X 0,Y 488.691,Z 254.423,A -85,B 0,C 180,E1 -6681.072,E2 -6681.072} C_VEL
LIN {X 0,Y 488.666,Z 254.428,A -85,B 0,C 180,E1 -6683.747,E2 -6683.747} C_VEL
LIN {X 0,Y 488.682,Z 254.423,A -85,B 0,C 180,E1 -6686.476,E2 -6686.476} C_VEL
LIN {X 0,Y 488.688,Z 254.426,A -85,B 0,C 180,E1 -6689.273,E2 -6689.273} C_VEL
LIN {X 0,Y 488.696,Z 254.422,A -85,B 0,C 180,E1 -6692.148,E2 -6692.148} C_VEL
LIN {X 0,Y 488.711,Z 254.423,A -85,B 0,C 180,E1 -6695.116,E2 -6695.116} C_VEL
LIN {X 0,Y 488.663,Z 254.426,A -85,B 0,C 180,E1 -6698.202,E2 -6698.202} C_VEL
LIN {X 0,Y 488.695,Z 254.422,A -85,B 0,C 180,E1 -6700.341,E2 -6700.341} C_VEL
LIN {X 0,Y 488.674,Z 254.427,A -85,B 0,C 180,E1 -6703.656,E2 -6703.656} C_VEL
LIN {X 0,Y 488.674,Z 254.424,A -85,B 0,C 180,E1 -6706.344,E2 -6706.344} C_VEL
LIN {X 0,Y 488.705,Z 254.422,A -85,B 0,C 180,E1 -6709.673,E2 -6709.673} C_VEL
LIN {X 0,Y 488.671,Z 254.427,A -85,B 0,C 180,E1 -6712.84,E2 -6712.84} C_VEL
LIN {X 0,Y 488.719,Z 254.419,A -85,B 0,C 180,E1 -6715.886,E2 -6715.886} C_VEL
LIN {X 0,Y 488.672,Z 254.427,A -85,B 0,C 180,E1 -6718.818,E2 -6718.818} C_VEL
LIN {X 0,Y 488.694,Z 254.422,A -85,B 0,C 180,E1 -6721.668,E2 -6721.668} C_VEL
LIN {X 0,Y 488.682,Z 254.424,A -85,B 0,C 180,E1 -6724.3,E2 -6724.3} C_VEL
LIN {X 0,Y 488.048,Z 254.507,A -85,B 0,C 180,E1 -6724.988,E2 -6724.988} C_VEL
LIN {X 0,Y 485.201,Z 254.862,A -85,B 0,C 180,E1 -6726.105,E2 -6726.105} C_VEL
LIN {X 0,Y 482.769,Z 255.164,A -85,B 0,C 180,E1 -6727.006,E2 -6727.006} C_VEL
LIN {X 0,Y 481.718,Z 255.291,A -85,B 0,C 180,E1 -6727.701,E2 -6727.701} C_VEL
LIN {X 0,Y 481.63,Z 255.301,A -85,B 0,C 180,E1 -6727.937,E2 -6727.937} C_VEL
LIN {X 0,Y 481.697,Z 255.298,A -85,B 0,C 180,E1 -6730.392,E2 -6730.392} C_VEL
LIN {X 0,Y 481.614,Z 255.308,A -85,B 0,C 180,E1 -6733.031,E2 -6733.031} C_VEL
LIN {X 0,Y 481.568,Z 255.472,A -85,B 0,C 180,E1 -6734.362,E2 -6734.362} C_VEL
LIN {X 0,Y 481.52,Z 267.629,A -85,B 0,C 180,E1 -6737.074,E2 -6737.074} C_VEL
LIN {X 0,Y 483.507,Z 279.079,A -85,B 0,C 180,E1 -6737.303,E2 -6737.303} C_VEL
LIN {X 0,Y 483.065,Z 343.51,A -85,B 0,C 180,E1 -6738.274,E2 -6738.274} C_VEL
LIN {X 0,Y 482.944,Z 352.641,A -85,B 0,C 180,E1 -6738.51,E2 -6738.51} C_VEL
LIN {X 0,Y 482.806,Z 362.238,A -85,B 0,C 180,E1 -6738.879,E2 -6738.879} C_VEL
LIN {X 0,Y 482.617,Z 372.269,A -85,B 0,C 180,E1 -6739.406,E2 -6739.406} C_VEL
LIN {X 0,Y 482.4,Z 382.671,A -85,B 0,C 180,E1 -6740.143,E2 -6740.143} C_VEL
LIN {X 0,Y 482.082,Z 390.798,A -85,B 0,C 180,E1 -6740.877,E2 -6740.877} C_VEL
LIN {X 0,Y 481.819,Z 397.498,A -85,B 0,C 180,E1 -6741.612,E2 -6741.612} C_VEL
LIN {X 0,Y 481.614,Z 403.835,A -85,B 0,C 180,E1 -6742.453,E2 -6742.453} C_VEL
LIN {X 0,Y 481.509,Z 409.097,A -85,B 0,C 180,E1 -6743.294,E2 -6743.294} C_VEL
LIN {X 0,Y 481.224,Z 413.5,A -85,B 0,C 180,E1 -6744.132,E2 -6744.132} C_VEL
LIN {X 0,Y 481.245,Z 417.152,A -85,B 0,C 180,E1 -6744.973,E2 -6744.973} C_VEL
LIN {X 0,Y 481.109,Z 420.14,A -85,B 0,C 180,E1 -6745.811,E2 -6745.811} C_VEL
LIN {X 0,Y 481.082,Z 422.45,A -85,B 0,C 180,E1 -6746.65,E2 -6746.65} C_VEL
LIN {X 0,Y 480.956,Z 424.217,A -85,B 0,C 180,E1 -6747.487,E2 -6747.487} C_VEL
LIN {X 0,Y 480.832,Z 425.494,A -85,B 0,C 180,E1 -6748.324,E2 -6748.324} C_VEL
LIN {X 0,Y 480.778,Z 426.302,A -85,B 0,C 180,E1 -6749.162,E2 -6749.162} C_VEL
LIN {X 0,Y 480.768,Z 426.609,A -85,B 0,C 180,E1 -6750,E2 -6750} C_VEL
LIN {X 0,Y 480.778,Z 426.336,A -85,B 0,C 180,E1 -6750.837,E2 -6750.837} C_VEL
LIN {X 0,Y 480.833,Z 425.599,A -85,B 0,C 180,E1 -6751.675,E2 -6751.675} C_VEL
LIN {X 0,Y 480.956,Z 424.393,A -85,B 0,C 180,E1 -6752.512,E2 -6752.512} C_VEL
LIN {X 0,Y 481.087,Z 421.561,A -85,B 0,C 180,E1 -6753.769,E2 -6753.769} C_VEL
LIN {X 0,Y 481.169,Z 418.985,A -85,B 0,C 180,E1 -6754.607,E2 -6754.607} C_VEL
LIN {X 0,Y 481.218,Z 413.916,A -85,B 0,C 180,E1 -6755.867,E2 -6755.867} C_VEL
LIN {X 0,Y 481.502,Z 409.609,A -85,B 0,C 180,E1 -6756.705,E2 -6756.705} C_VEL
LIN {X 0,Y 481.618,Z 403.043,A -85,B 0,C 180,E1 -6757.757,E2 -6757.757} C_VEL
LIN {X 0,Y 481.983,Z 394.716,A -85,B 0,C 180,E1 -6758.806,E2 -6758.806} C_VEL
LIN {X 0,Y 482.281,Z 386.177,A -85,B 0,C 180,E1 -6759.647,E2 -6759.647} C_VEL
LIN {X 0,Y 482.423,Z 378.296,A -85,B 0,C 180,E1 -6760.28,E2 -6760.28} C_VEL
LIN {X 0,Y 482.683,Z 370.15,A -85,B 0,C 180,E1 -6760.804,E2 -6760.804} C_VEL
LIN {X 0,Y 482.883,Z 361.905,A -85,B 0,C 180,E1 -6761.225,E2 -6761.225} C_VEL
LIN {X 0,Y 482.956,Z 353.016,A -85,B 0,C 180,E1 -6761.568,E2 -6761.568} C_VEL
LIN {X 0,Y 483.144,Z 343.69,A -85,B 0,C 180,E1 -6761.811,E2 -6761.811} C_VEL
LIN {X 0,Y 483.404,Z 278.125,A -85,B 0,C 180,E1 -6762.805,E2 -6762.805} C_VEL
LIN {X 0,Y 481.506,Z 267.583,A -85,B 0,C 180,E1 -6763.03,E2 -6763.03} C_VEL
LIN {X 0,Y 481.511,Z 255.325,A -85,B 0,C 180,E1 -6765.771,E2 -6765.771} C_VEL
LIN {X 0,Y 481.703,Z 255.293,A -85,B 0,C 180,E1 -6768.722,E2 -6768.722} C_VEL
LIN {X 0,Y 481.638,Z 255.304,A -85,B 0,C 180,E1 -6771.394,E2 -6771.394} C_VEL
LIN {X 0,Y 481.644,Z 255.3,A -85,B 0,C 180,E1 -6774.114,E2 -6774.114} C_VEL
LIN {X 0,Y 481.65,Z 255.303,A -85,B 0,C 180,E1 -6777.116,E2 -6777.116} C_VEL
LIN {X 0,Y 481.649,Z 255.301,A -85,B 0,C 180,E1 -6779.742,E2 -6779.742} C_VEL
LIN {X 0,Y 481.647,Z 255.302,A -85,B 0,C 180,E1 -6782.675,E2 -6782.675} C_VEL
LIN {X 0,Y 481.625,Z 255.304,A -85,B 0,C 180,E1 -6785.71,E2 -6785.71} C_VEL
LIN {X 0,Y 481.662,Z 255.301,A -85,B 0,C 180,E1 -6788.859,E2 -6788.859} C_VEL
LIN {X 0,Y 481.612,Z 255.305,A -85,B 0,C 180,E1 -6792.164,E2 -6792.164} C_VEL
LIN {X 0,Y 481.65,Z 255.302,A -85,B 0,C 180,E1 -6794.458,E2 -6794.458} C_VEL
LIN {X 0,Y 481.611,Z 255.307,A -85,B 0,C 180,E1 -6796.855,E2 -6796.855} C_VEL
LIN {X 0,Y 481.651,Z 255.3,A -85,B 0,C 180,E1 -6800.057,E2 -6800.057} C_VEL
LIN {X 0,Y 481.613,Z 255.306,A -85,B 0,C 180,E1 -6803.252,E2 -6803.252} C_VEL
LIN {X 0,Y 481.666,Z 255.301,A -85,B 0,C 180,E1 -6806.326,E2 -6806.326} C_VEL
LIN {X 0,Y 481.629,Z 255.302,A -85,B 0,C 180,E1 -6809.421,E2 -6809.421} C_VEL
LIN {X 0,Y 481.642,Z 255.304,A -85,B 0,C 180,E1 -6812.164,E2 -6812.164} C_VEL
LIN {X 0,Y 481.668,Z 255.299,A -85,B 0,C 180,E1 -6814.967,E2 -6814.967} C_VEL
LIN {X 0,Y 481.63,Z 255.303,A -85,B 0,C 180,E1 -6817.704,E2 -6817.704} C_VEL
LIN {X 0,Y 481.687,Z 255.298,A -85,B 0,C 180,E1 -6820.392,E2 -6820.392} C_VEL
LIN {X 0,Y 481.616,Z 255.304,A -85,B 0,C 180,E1 -6823.031,E2 -6823.031} C_VEL
LIN {X 0,Y 481.666,Z 255.299,A -85,B 0,C 180,E1 -6825.638,E2 -6825.638} C_VEL
LIN {X 0,Y 481.729,Z 255.292,A -85,B 0,C 180,E1 -6828.214,E2 -6828.214} C_VEL
LIN {X 0,Y 481.71,Z 255.294,A -85,B 0,C 180,E1 -6831.611,E2 -6831.611} C_VEL
LIN {X 0,Y 481.769,Z 255.288,A -85,B 0,C 180,E1 -6834.139,E2 -6834.139} C_VEL
LIN {X 0,Y 481.9,Z 255.27,A -85,B 0,C 180,E1 -6837.492,E2 -6837.492} C_VEL
LIN {X 0,Y 481.904,Z 255.271,A -85,B 0,C 180,E1 -6840,E2 -6840} C_VEL
LIN {X 0,Y 481.9,Z 255.269,A -85,B 0,C 180,E1 -6842.508,E2 -6842.508} C_VEL
LIN {X 0,Y 481.765,Z 255.288,A -85,B 0,C 180,E1 -6845.861,E2 -6845.861} C_VEL
LIN {X 0,Y 481.709,Z 255.293,A -85,B 0,C 180,E1 -6848.389,E2 -6848.389} C_VEL
LIN {X 0,Y 481.729,Z 255.294,A -85,B 0,C 180,E1 -6851.785,E2 -6851.785} C_VEL
LIN {X 0,Y 481.722,Z 255.292,A -85,B 0,C 180,E1 -6855.225,E2 -6855.225} C_VEL
LIN {X 0,Y 481.643,Z 255.3,A -85,B 0,C 180,E1 -6858.724,E2 -6858.724} C_VEL
LIN {X 0,Y 481.623,Z 255.306,A -85,B 0,C 180,E1 -6861.396,E2 -6861.396} C_VEL
LIN {X 0,Y 481.635,Z 255.301,A -85,B 0,C 180,E1 -6864.115,E2 -6864.115} C_VEL
LIN {X 0,Y 481.644,Z 255.302,A -85,B 0,C 180,E1 -6867.117,E2 -6867.117} C_VEL
LIN {X 0,Y 481.594,Z 255.308,A -85,B 0,C 180,E1 -6869.747,E2 -6869.747} C_VEL
LIN {X 0,Y 481.643,Z 255.3,A -85,B 0,C 180,E1 -6872.676,E2 -6872.676} C_VEL
LIN {X 0,Y 481.644,Z 255.304,A -85,B 0,C 180,E1 -6875.202,E2 -6875.202} C_VEL
LIN {X 0,Y 481.624,Z 255.301,A -85,B 0,C 180,E1 -6878.004,E2 -6878.004} C_VEL
LIN {X 0,Y 481.617,Z 255.308,A -85,B 0,C 180,E1 -6881.046,E2 -6881.046} C_VEL
LIN {X 0,Y 481.648,Z 255.299,A -85,B 0,C 180,E1 -6884.459,E2 -6884.459} C_VEL
LIN {X 0,Y 481.609,Z 255.303,A -85,B 0,C 180,E1 -6887.836,E2 -6887.836} C_VEL
LIN {X 0,Y 481.642,Z 255.303,A -85,B 0,C 180,E1 -6890.657,E2 -6890.657} C_VEL
LIN {X 0,Y 481.602,Z 255.305,A -85,B 0,C 180,E1 -6893.38,E2 -6893.38} C_VEL
LIN {X 0,Y 481.667,Z 255.297,A -85,B 0,C 180,E1 -6896.327,E2 -6896.327} C_VEL
LIN {X 0,Y 481.606,Z 255.303,A -85,B 0,C 180,E1 -6899.426,E2 -6899.426} C_VEL
LIN {X 0,Y 481.638,Z 255.303,A -85,B 0,C 180,E1 -6902.165,E2 -6902.165} C_VEL
LIN {X 0,Y 481.678,Z 255.363,A -85,B 0,C 180,E1 -6905.515,E2 -6905.515} C_VEL
LIN {X 0,Y 482.985,Z 263.526,A -85,B 0,C 180,E1 -6907.093,E2 -6907.093} C_VEL
LIN {X 0,Y 482.516,Z 279.321,A -85,B 0,C 180,E1 -6909.984,E2 -6909.984} C_VEL
LIN {X 0,Y 482.074,Z 293.844,A -85,B 0,C 180,E1 -6912.611,E2 -6912.611} C_VEL
LIN {X 0,Y 481.678,Z 310.724,A -85,B 0,C 180,E1 -6915.639,E2 -6915.639} C_VEL
LIN {X 0,Y 481.506,Z 318.427,A -85,B 0,C 180,E1 -6917.013,E2 -6917.013} C_VEL
LIN {X 0,Y 483.25,Z 335.219,A -85,B 0,C 180,E1 -6917.311,E2 -6917.311} C_VEL
LIN {X 0,Y 482.91,Z 396.705,A -85,B 0,C 180,E1 -6918.244,E2 -6918.244} C_VEL
LIN {X 0,Y 482.679,Z 407.174,A -85,B 0,C 180,E1 -6918.531,E2 -6918.531} C_VEL
LIN {X 0,Y 482.457,Z 417.9,A -85,B 0,C 180,E1 -6918.978,E2 -6918.978} C_VEL
LIN {X 0,Y 482.079,Z 428.548,A -85,B 0,C 180,E1 -6919.607,E2 -6919.607} C_VEL
LIN {X 0,Y 481.854,Z 436.897,A -85,B 0,C 180,E1 -6920.239,E2 -6920.239} C_VEL
LIN {X 0,Y 481.581,Z 444.799,A -85,B 0,C 180,E1 -6920.975,E2 -6920.975} C_VEL
LIN {X 0,Y 481.361,Z 452.194,A -85,B 0,C 180,E1 -6921.816,E2 -6921.816} C_VEL
LIN {X 0,Y 481.202,Z 459.702,A -85,B 0,C 180,E1 -6922.869,E2 -6922.869} C_VEL
LIN {X 0,Y 480.992,Z 466.56,A -85,B 0,C 180,E1 -6924.13,E2 -6924.13} C_VEL
LIN {X 0,Y 480.873,Z 471.768,A -85,B 0,C 180,E1 -6925.39,E2 -6925.39} C_VEL
LIN {X 0,Y 480.916,Z 475.6,A -85,B 0,C 180,E1 -6926.649,E2 -6926.649} C_VEL
LIN {X 0,Y 480.872,Z 477.36,A -85,B 0,C 180,E1 -6927.487,E2 -6927.487} C_VEL
LIN {X 0,Y 480.823,Z 478.62,A -85,B 0,C 180,E1 -6928.325,E2 -6928.325} C_VEL
LIN {X 0,Y 480.766,Z 479.403,A -85,B 0,C 180,E1 -6929.163,E2 -6929.163} C_VEL
LIN {X 0,Y 480.759,Z 479.699,A -85,B 0,C 180,E1 -6930,E2 -6930} C_VEL
LIN {X 0,Y 480.766,Z 479.402,A -85,B 0,C 180,E1 -6930.838,E2 -6930.838} C_VEL
LIN {X 0,Y 480.823,Z 478.618,A -85,B 0,C 180,E1 -6931.676,E2 -6931.676} C_VEL
LIN {X 0,Y 480.872,Z 477.357,A -85,B 0,C 180,E1 -6932.513,E2 -6932.513} C_VEL
LIN {X 0,Y 480.938,Z 474.434,A -85,B 0,C 180,E1 -6933.771,E2 -6933.771} C_VEL
LIN {X 0,Y 480.874,Z 471.764,A -85,B 0,C 180,E1 -6934.611,E2 -6934.611} C_VEL
LIN {X 0,Y 480.992,Z 466.551,A -85,B 0,C 180,E1 -6935.871,E2 -6935.871} C_VEL
LIN {X 0,Y 481.168,Z 459.686,A -85,B 0,C 180,E1 -6937.132,E2 -6937.132} C_VEL
LIN {X 0,Y 481.362,Z 452.185,A -85,B 0,C 180,E1 -6938.184,E2 -6938.184} C_VEL
LIN {X 0,Y 481.582,Z 444.792,A -85,B 0,C 180,E1 -6939.026,E2 -6939.026} C_VEL
LIN {X 0,Y 481.855,Z 436.883,A -85,B 0,C 180,E1 -6939.762,E2 -6939.762} C_VEL
LIN {X 0,Y 482.08,Z 428.528,A -85,B 0,C 180,E1 -6940.394,E2 -6940.394} C_VEL
LIN {X 0,Y 482.454,Z 417.874,A -85,B 0,C 180,E1 -6941.023,E2 -6941.023} C_VEL
LIN {X 0,Y 482.682,Z 406.294,A -85,B 0,C 180,E1 -6941.496,E2 -6941.496} C_VEL
LIN {X 0,Y 482.938,Z 396.629,A -85,B 0,C 180,E1 -6941.756,E2 -6941.756} C_VEL
LIN {X 0,Y 483.273,Z 334.634,A -85,B 0,C 180,E1 -6942.696,E2 -6942.696} C_VEL
LIN {X 0,Y 481.504,Z 318.425,A -85,B 0,C 180,E1 -6942.987,E2 -6942.987} C_VEL
LIN {X 0,Y 481.841,Z 302.698,A -85,B 0,C 180,E1 -6945.797,E2 -6945.797} C_VEL
LIN {X 0,Y 482.383,Z 285.491,A -85,B 0,C 180,E1 -6948.893,E2 -6948.893} C_VEL
LIN {X 0,Y 482.845,Z 268.377,A -85,B 0,C 180,E1 -6952.012,E2 -6952.012} C_VEL
LIN {X 0,Y 482.861,Z 262.28,A -85,B 0,C 180,E1 -6953.141,E2 -6953.141} C_VEL
LIN {X 0,Y 481.681,Z 255.296,A -85,B 0,C 180,E1 -6954.515,E2 -6954.515} C_VEL
LIN {X 0,Y 481.641,Z 255.301,A -85,B 0,C 180,E1 -6957.836,E2 -6957.836} C_VEL
LIN {X 0,Y 481.608,Z 255.303,A -85,B 0,C 180,E1 -6960.714,E2 -6960.714} C_VEL
LIN {X 0,Y 481.649,Z 255.299,A -85,B 0,C 180,E1 -6963.725,E2 -6963.725} C_VEL
LIN {X 0,Y 481.6,Z 255.306,A -85,B 0,C 180,E1 -6966.75,E2 -6966.75} C_VEL
LIN {X 0,Y 481.628,Z 255.301,A -85,B 0,C 180,E1 -6969.946,E2 -6969.946} C_VEL
LIN {X 0,Y 481.614,Z 255.306,A -85,B 0,C 180,E1 -6973.303,E2 -6973.303} C_VEL
LIN {X 0,Y 481.648,Z 255.299,A -85,B 0,C 180,E1 -6975.642,E2 -6975.642} C_VEL
LIN {X 0,Y 481.612,Z 255.308,A -85,B 0,C 180,E1 -6978.954,E2 -6978.954} C_VEL
LIN {X 0,Y 481.626,Z 255.301,A -85,B 0,C 180,E1 -6981.998,E2 -6981.998} C_VEL
LIN {X 0,Y 481.672,Z 255.297,A -85,B 0,C 180,E1 -6985.317,E2 -6985.317} C_VEL
LIN {X 0,Y 481.62,Z 255.305,A -85,B 0,C 180,E1 -6988.31,E2 -6988.31} C_VEL
LIN {X 0,Y 481.633,Z 255.302,A -85,B 0,C 180,E1 -6991.214,E2 -6991.214} C_VEL
LIN {X 0,Y 481.618,Z 255.304,A -85,B 0,C 180,E1 -6994.038,E2 -6994.038} C_VEL
LIN {X 0,Y 481.634,Z 255.303,A -85,B 0,C 180,E1 -6996.824,E2 -6996.824} C_VEL
LIN {X 0,Y 481.618,Z 255.303,A -85,B 0,C 180,E1 -6999.499,E2 -6999.499} C_VEL
LIN {X 0,Y 481.646,Z 255.303,A -85,B 0,C 180,E1 -7002.156,E2 -7002.156} C_VEL
LIN {X 0,Y 481.69,Z 255.296,A -85,B 0,C 180,E1 -7004.774,E2 -7004.774} C_VEL
LIN {X 0,Y 481.726,Z 255.294,A -85,B 0,C 180,E1 -7008.215,E2 -7008.215} C_VEL
LIN {X 0,Y 481.713,Z 255.292,A -85,B 0,C 180,E1 -7011.611,E2 -7011.611} C_VEL
LIN {X 0,Y 481.772,Z 255.288,A -85,B 0,C 180,E1 -7014.139,E2 -7014.139} C_VEL
LIN {X 0,Y 481.906,Z 255.268,A -85,B 0,C 180,E1 -7017.493,E2 -7017.493} C_VEL
LIN {X 0,Y 481.91,Z 255.271,A -85,B 0,C 180,E1 -7020,E2 -7020} C_VEL
LIN {X 0,Y 481.906,Z 255.27,A -85,B 0,C 180,E1 -7022.508,E2 -7022.508} C_VEL
LIN {X 0,Y 481.772,Z 255.288,A -85,B 0,C 180,E1 -7025.861,E2 -7025.861} C_VEL
LIN {X 0,Y 481.713,Z 255.294,A -85,B 0,C 180,E1 -7028.389,E2 -7028.389} C_VEL
LIN {X 0,Y 481.736,Z 255.292,A -85,B 0,C 180,E1 -7031.785,E2 -7031.785} C_VEL
LIN {X 0,Y 481.73,Z 255.291,A -85,B 0,C 180,E1 -7035.225,E2 -7035.225} C_VEL
LIN {X 0,Y 481.65,Z 255.299,A -85,B 0,C 180,E1 -7038.724,E2 -7038.724} C_VEL
LIN {X 0,Y 481.63,Z 255.306,A -85,B 0,C 180,E1 -7041.396,E2 -7041.396} C_VEL
LIN {X 0,Y 481.646,Z 255.302,A -85,B 0,C 180,E1 -7044.115,E2 -7044.115} C_VEL
LIN {X 0,Y 481.652,Z 255.302,A -85,B 0,C 180,E1 -7047.117,E2 -7047.117} C_VEL
LIN {X 0,Y 481.654,Z 255.302,A -85,B 0,C 180,E1 -7049.743,E2 -7049.743} C_VEL
LIN {X 0,Y 481.652,Z 255.3,A -85,B 0,C 180,E1 -7052.676,E2 -7052.676} C_VEL
LIN {X 0,Y 481.629,Z 255.305,A -85,B 0,C 180,E1 -7055.71,E2 -7055.71} C_VEL
LIN {X 0,Y 481.658,Z 255.301,A -85,B 0,C 180,E1 -7058.86,E2 -7058.86} C_VEL
LIN {X 0,Y 481.622,Z 255.304,A -85,B 0,C 180,E1 -7061.908,E2 -7061.908} C_VEL
LIN {X 0,Y 481.655,Z 255.299,A -85,B 0,C 180,E1 -7064.458,E2 -7064.458} C_VEL
LIN {X 0,Y 481.616,Z 255.306,A -85,B 0,C 180,E1 -7066.855,E2 -7066.855} C_VEL
LIN {X 0,Y 481.658,Z 255.298,A -85,B 0,C 180,E1 -7070.057,E2 -7070.057} C_VEL
LIN {X 0,Y 481.621,Z 255.307,A -85,B 0,C 180,E1 -7073.252,E2 -7073.252} C_VEL
LIN {X 0,Y 481.672,Z 255.298,A -85,B 0,C 180,E1 -7076.327,E2 -7076.327} C_VEL
LIN {X 0,Y 481.629,Z 255.304,A -85,B 0,C 180,E1 -7079.422,E2 -7079.422} C_VEL
LIN {X 0,Y 481.651,Z 255.3,A -85,B 0,C 180,E1 -7082.165,E2 -7082.165} C_VEL
LIN {X 0,Y 481.675,Z 255.3,A -85,B 0,C 180,E1 -7084.967,E2 -7084.967} C_VEL
LIN {X 0,Y 481.63,Z 255.301,A -85,B 0,C 180,E1 -7087.937,E2 -7087.937} C_VEL
LIN {X 0,Y 480.966,Z 255.388,A -85,B 0,C 180,E1 -7088.635,E2 -7088.635} C_VEL
LIN {X 0,Y 478.15,Z 255.735,A -85,B 0,C 180,E1 -7089.769,E2 -7089.769} C_VEL
LIN {X 0,Y 475.764,Z 256.04,A -85,B 0,C 180,E1 -7090.684,E2 -7090.684} C_VEL
LIN {X 0,Y 474.731,Z 256.162,A -85,B 0,C 180,E1 -7091.39,E2 -7091.39} C_VEL
LIN {X 0,Y 474.642,Z 256.172,A -85,B 0,C 180,E1 -7091.629,E2 -7091.629} C_VEL
LIN {X 0,Y 474.526,Z 256.278,A -85,B 0,C 180,E1 -7094.255,E2 -7094.255} C_VEL
LIN {X 0,Y 474.55,Z 268.148,A -85,B 0,C 180,E1 -7096.885,E2 -7096.885} C_VEL
LIN {X 0,Y 476.611,Z 280.483,A -85,B 0,C 180,E1 -7097.131,E2 -7097.131} C_VEL
LIN {X 0,Y 476.13,Z 343.923,A -85,B 0,C 180,E1 -7098.101,E2 -7098.101} C_VEL
LIN {X 0,Y 476.008,Z 353.046,A -85,B 0,C 180,E1 -7098.341,E2 -7098.341} C_VEL
LIN {X 0,Y 475.864,Z 362.639,A -85,B 0,C 180,E1 -7098.715,E2 -7098.715} C_VEL
LIN {X 0,Y 475.661,Z 372.668,A -85,B 0,C 180,E1 -7099.249,E2 -7099.249} C_VEL
LIN {X 0,Y 475.438,Z 383.067,A -85,B 0,C 180,E1 -7099.997,E2 -7099.997} C_VEL
LIN {X 0,Y 475.112,Z 391.192,A -85,B 0,C 180,E1 -7100.742,E2 -7100.742} C_VEL
LIN {X 0,Y 474.822,Z 397.893,A -85,B 0,C 180,E1 -7101.488,E2 -7101.488} C_VEL
LIN {X 0,Y 474.59,Z 404.229,A -85,B 0,C 180,E1 -7102.341,E2 -7102.341} C_VEL
LIN {X 0,Y 474.477,Z 409.49,A -85,B 0,C 180,E1 -7103.194,E2 -7103.194} C_VEL
LIN {X 0,Y 474.191,Z 413.893,A -85,B 0,C 180,E1 -7104.045,E2 -7104.045} C_VEL
LIN {X 0,Y 474.135,Z 419.048,A -85,B 0,C 180,E1 -7105.323,E2 -7105.323} C_VEL
LIN {X 0,Y 474.016,Z 421.704,A -85,B 0,C 180,E1 -7106.174,E2 -7106.174} C_VEL
LIN {X 0,Y 473.9,Z 424.608,A -85,B 0,C 180,E1 -7107.45,E2 -7107.45} C_VEL
LIN {X 0,Y 473.767,Z 425.885,A -85,B 0,C 180,E1 -7108.299,E2 -7108.299} C_VEL
LIN {X 0,Y 473.705,Z 426.692,A -85,B 0,C 180,E1 -7109.149,E2 -7109.149} C_VEL
LIN {X 0,Y 473.693,Z 426.999,A -85,B 0,C 180,E1 -7110,E2 -7110} C_VEL
LIN {X 0,Y 473.706,Z 426.727,A -85,B 0,C 180,E1 -7110.85,E2 -7110.85} C_VEL
LIN {X 0,Y 473.767,Z 425.989,A -85,B 0,C 180,E1 -7111.7,E2 -7111.7} C_VEL
LIN {X 0,Y 473.9,Z 424.782,A -85,B 0,C 180,E1 -7112.55,E2 -7112.55} C_VEL
LIN {X 0,Y 474.013,Z 421.951,A -85,B 0,C 180,E1 -7113.825,E2 -7113.825} C_VEL
LIN {X 0,Y 474.12,Z 419.374,A -85,B 0,C 180,E1 -7114.676,E2 -7114.676} C_VEL
LIN {X 0,Y 474.185,Z 414.304,A -85,B 0,C 180,E1 -7115.955,E2 -7115.955} C_VEL
LIN {X 0,Y 474.498,Z 408.486,A -85,B 0,C 180,E1 -7117.083,E2 -7117.083} C_VEL
LIN {X 0,Y 474.705,Z 401.975,A -85,B 0,C 180,E1 -7118.085,E2 -7118.085} C_VEL
LIN {X 0,Y 475.002,Z 394.089,A -85,B 0,C 180,E1 -7119.044,E2 -7119.044} C_VEL
LIN {X 0,Y 475.301,Z 386.563,A -85,B 0,C 180,E1 -7119.79,E2 -7119.79} C_VEL
LIN {X 0,Y 475.468,Z 378.68,A -85,B 0,C 180,E1 -7120.432,E2 -7120.432} C_VEL
LIN {X 0,Y 475.738,Z 370.533,A -85,B 0,C 180,E1 -7120.964,E2 -7120.964} C_VEL
LIN {X 0,Y 475.948,Z 362.285,A -85,B 0,C 180,E1 -7121.39,E2 -7121.39} C_VEL
LIN {X 0,Y 476.031,Z 353.392,A -85,B 0,C 180,E1 -7121.739,E2 -7121.739} C_VEL
LIN {X 0,Y 476.204,Z 344.19,A -85,B 0,C 180,E1 -7121.983,E2 -7121.983} C_VEL
LIN {X 0,Y 476.456,Z 278.689,A -85,B 0,C 180,E1 -7122.992,E2 -7122.992} C_VEL
LIN {X 0,Y 474.503,Z 267.934,A -85,B 0,C 180,E1 -7123.225,E2 -7123.225} C_VEL
LIN {X 0,Y 474.478,Z 256.201,A -85,B 0,C 180,E1 -7125.874,E2 -7125.874} C_VEL
LIN {X 0,Y 474.655,Z 256.171,A -85,B 0,C 180,E1 -7128.627,E2 -7128.627} C_VEL
LIN {X 0,Y 474.58,Z 256.182,A -85,B 0,C 180,E1 -7131.729,E2 -7131.729} C_VEL
LIN {X 0,Y 474.623,Z 256.175,A -85,B 0,C 180,E1 -7134.494,E2 -7134.494} C_VEL
LIN {X 0,Y 474.596,Z 256.18,A -85,B 0,C 180,E1 -7137.326,E2 -7137.326} C_VEL
LIN {X 0,Y 474.578,Z 256.18,A -85,B 0,C 180,E1 -7140.231,E2 -7140.231} C_VEL
LIN {X 0,Y 474.611,Z 256.178,A -85,B 0,C 180,E1 -7143.222,E2 -7143.222} C_VEL
LIN {X 0,Y 474.579,Z 256.181,A -85,B 0,C 180,E1 -7146.324,E2 -7146.324} C_VEL
LIN {X 0,Y 474.618,Z 256.177,A -85,B 0,C 180,E1 -7149.548,E2 -7149.548} C_VEL
LIN {X 0,Y 474.572,Z 256.182,A -85,B 0,C 180,E1 -7152.23,E2 -7152.23} C_VEL
LIN {X 0,Y 474.612,Z 256.179,A -85,B 0,C 180,E1 -7155.297,E2 -7155.297} C_VEL
LIN {X 0,Y 474.587,Z 256.181,A -85,B 0,C 180,E1 -7158.211,E2 -7158.211} C_VEL
LIN {X 0,Y 474.597,Z 256.179,A -85,B 0,C 180,E1 -7161.541,E2 -7161.541} C_VEL
LIN {X 0,Y 474.612,Z 256.178,A -85,B 0,C 180,E1 -7164.724,E2 -7164.724} C_VEL
LIN {X 0,Y 474.621,Z 256.176,A -85,B 0,C 180,E1 -7167.786,E2 -7167.786} C_VEL
LIN {X 0,Y 474.588,Z 256.183,A -85,B 0,C 180,E1 -7170.891,E2 -7170.891} C_VEL
LIN {X 0,Y 474.584,Z 256.18,A -85,B 0,C 180,E1 -7173.624,E2 -7173.624} C_VEL
LIN {X 0,Y 474.628,Z 256.177,A -85,B 0,C 180,E1 -7176.642,E2 -7176.642} C_VEL
LIN {X 0,Y 474.636,Z 256.175,A -85,B 0,C 180,E1 -7180.089,E2 -7180.089} C_VEL
LIN {X 0,Y 474.59,Z 256.181,A -85,B 0,C 180,E1 -7182.772,E2 -7182.772} C_VEL
LIN {X 0,Y 474.625,Z 256.175,A -85,B 0,C 180,E1 -7185.42,E2 -7185.42} C_VEL
LIN {X 0,Y 474.687,Z 256.169,A -85,B 0,C 180,E1 -7188.037,E2 -7188.037} C_VEL
LIN {X 0,Y 474.658,Z 256.172,A -85,B 0,C 180,E1 -7191.485,E2 -7191.485} C_VEL
LIN {X 0,Y 474.732,Z 256.164,A -85,B 0,C 180,E1 -7194.052,E2 -7194.052} C_VEL
LIN {X 0,Y 474.865,Z 256.146,A -85,B 0,C 180,E1 -7197.455,E2 -7197.455} C_VEL
LIN {X 0,Y 474.873,Z 256.147,A -85,B 0,C 180,E1 -7200,E2 -7200} C_VEL
LIN {X 0,Y 474.865,Z 256.145,A -85,B 0,C 180,E1 -7202.545,E2 -7202.545} C_VEL
LIN {X 0,Y 474.729,Z 256.165,A -85,B 0,C 180,E1 -7205.948,E2 -7205.948} C_VEL
LIN {X 0,Y 474.658,Z 256.171,A -85,B 0,C 180,E1 -7208.515,E2 -7208.515} C_VEL
LIN {X 0,Y 474.687,Z 256.171,A -85,B 0,C 180,E1 -7211.963,E2 -7211.963} C_VEL
